SPLINE
SPL {X  -133.093, Y  +296.896, Z    +0.000, E1   +44.059, E3 +170338.505}
SPL {X  -150.601, Y  +331.670, Z    +0.000, E1   +33.435, E3 +170362.768}
SPL {X  -157.739, Y  +358.898, Z    +0.000, E1   +20.026, E3 +170370.995}
SPL {X  -159.601, Y  +374.403, Z    +0.000, E1   +10.058, E3 +170373.311}
SPL {X  -159.993, Y  +384.251, Z    +0.000, E1    +2.830, E3 +170373.943}
SPL {X  -160.000, Y  +387.929, Z    +0.000, E1    -0.363, E3 +170374.011}
SPL {X  -160.000, Y  +392.137, Z    +0.000, E1    -6.580, E3 +170374.150}
SPL {X  -160.000, Y  +398.334, Z    +0.000, E1   -17.404, E3 +170374.642}
SPL {X  -160.000, Y  +410.558, Z    +0.000, E1   -36.649, E3 +170376.745}
SPL {X  -160.000, Y  +459.534, Z    +0.000, E1   -61.429, E3 +170396.339}
SPL {X  -160.000, Y  +586.246, Z    +0.000, E1   -66.315, E3 +170482.839}
SPL {X  -160.000, Y  +602.823, Z    +0.000, E1   -66.332, E3 +170498.243}
SPL {X  -160.000, Y  +621.796, Z    +0.000, E1   -66.332, E3 +170515.912}
SPL {X  -160.000, Y  +638.226, Z    +0.000, E1   -66.314, E3 +170531.239}
SPL {X  -160.000, Y  +655.092, Z    +0.000, E1   -66.336, E3 +170546.898}
SPL {X  -160.000, Y  +671.716, Z    +0.000, E1   -66.315, E3 +170562.412}
SPL {X  -159.502, Y  +687.017, Z    +0.000, E1   -66.266, E3 +170577.162}
SPL {X  -157.713, Y  +701.353, Z    +0.000, E1   -66.026, E3 +170592.389}
SPL {X  -155.081, Y  +713.767, Z    +0.000, E1   -65.665, E3 +170606.674}
SPL {X  -152.128, Y  +723.968, Z    +0.000, E1   -65.242, E3 +170619.174}
SPL {X  -148.925, Y  +732.892, Z    +0.000, E1   -64.779, E3 +170630.674}
SPL {X  -144.887, Y  +742.280, Z    +0.000, E1   -64.184, E3 +170643.303}
SPL {X  -140.317, Y  +751.285, Z    +0.000, E1   -63.454, E3 +170655.941}
SPL {X  -135.706, Y  +759.158, Z    +0.000, E1   -62.682, E3 +170667.342}
SPL {X  -131.040, Y  +766.207, Z    +0.000, E1   -61.854, E3 +170677.774}
SPL {X  -102.962, Y  +796.870, Z    +0.000, E1   -51.620, E3 +170803.106}
ENDSPLINE

SPLINE
SPL {X  -139.855, Y  +752.122, Z    +0.000, E1   -42.075, E3 +170926.034}
SPL {X  -153.268, Y  +720.324, Z    +0.000, E1   -30.648, E3 +170942.280}
SPL {X  -158.910, Y  +693.048, Z    +0.000, E1   -15.531, E3 +170948.350}
SPL {X  -159.977, Y  +677.095, Z    +0.000, E1    -3.968, E3 +170949.774}
SPL {X  -160.000, Y  +672.556, Z    +0.000, E1    -0.073, E3 +170949.876}
SPL {X  -160.000, Y  +669.399, Z    +0.000, E1    +3.976, E3 +170949.956}
SPL {X  -160.000, Y  +661.045, Z    +0.000, E1   +19.300, E3 +170950.544}
SPL {X  -160.000, Y  +646.999, Z    +0.000, E1   +41.048, E3 +170952.962}
SPL {X  -160.000, Y  +594.464, Z    +0.000, E1   +63.651, E3 +170973.262}
SPL {X  -160.000, Y  +465.200, Z    +0.000, E1   +67.027, E3 +171061.832}
SPL {X  -160.000, Y  +444.745, Z    +0.000, E1   +67.032, E3 +171080.241}
SPL {X  -160.000, Y  +422.224, Z    +0.000, E1   +67.044, E3 +171100.493}
ENDSPLINE

SPLINE
SPL {X  -160.000, Y  +424.635, Z    +0.000, E1   +64.425, E3 +171118.519}
ENDSPLINE

SPLINE
SPL {X  -160.000, Y  +410.501, Z    +0.000, E1   +64.162, E3 +171135.064}
SPL {X  -160.000, Y  +387.965, Z    +0.000, E1   +65.039, E3 +171151.016}
SPL {X  -158.836, Y  +366.435, Z    +0.000, E1   +65.805, E3 +171165.957}
SPL {X  -155.922, Y  +349.806, Z    +0.000, E1   +65.927, E3 +171180.603}
SPL {X  -152.875, Y  +338.486, Z    +0.000, E1   +65.488, E3 +171194.220}
SPL {X  -149.360, Y  +328.327, Z    +0.000, E1   +64.994, E3 +171207.126}
SPL {X  -145.195, Y  +318.481, Z    +0.000, E1   +64.365, E3 +171220.280}
SPL {X  -140.564, Y  +309.268, Z    +0.000, E1   +63.646, E3 +171233.101}
SPL {X  -135.770, Y  +301.044, Z    +0.000, E1   +62.840, E3 +171244.972}
SPL {X  -130.944, Y  +293.756, Z    +0.000, E1   +61.990, E3 +171255.715}
SPL {X  -103.957, Y  +264.074, Z    +0.000, E1   +52.557, E3 +171361.819}
ENDSPLINE

SPLINE
SPL {X  -133.093, Y  +296.896, Z    +0.000, E1   +44.059, E3 +171486.653}
SPL {X  -150.601, Y  +331.670, Z    +0.000, E1   +33.435, E3 +171510.915}
SPL {X  -157.739, Y  +358.898, Z    +0.000, E1   +20.026, E3 +171519.143}
SPL {X  -159.601, Y  +374.403, Z    +0.000, E1   +10.058, E3 +171521.459}
SPL {X  -159.993, Y  +384.251, Z    +0.000, E1    +2.830, E3 +171522.091}
SPL {X  -160.000, Y  +387.929, Z    +0.000, E1    -0.363, E3 +171522.159}
SPL {X  -160.000, Y  +392.137, Z    +0.000, E1    -6.580, E3 +171522.298}
SPL {X  -160.000, Y  +398.334, Z    +0.000, E1   -17.404, E3 +171522.790}
SPL {X  -160.000, Y  +410.558, Z    +0.000, E1   -36.649, E3 +171524.893}
SPL {X  -160.000, Y  +459.534, Z    +0.000, E1   -61.429, E3 +171544.487}
SPL {X  -160.000, Y  +586.246, Z    +0.000, E1   -66.315, E3 +171630.987}
SPL {X  -160.000, Y  +602.823, Z    +0.000, E1   -66.332, E3 +171646.391}
SPL {X  -160.000, Y  +621.796, Z    +0.000, E1   -66.332, E3 +171664.060}
SPL {X  -160.000, Y  +638.226, Z    +0.000, E1   -66.314, E3 +171679.387}
SPL {X  -160.000, Y  +655.092, Z    +0.000, E1   -66.336, E3 +171695.046}
SPL {X  -160.000, Y  +671.716, Z    +0.000, E1   -66.315, E3 +171710.560}
SPL {X  -159.502, Y  +687.017, Z    +0.000, E1   -66.266, E3 +171725.310}
SPL {X  -157.713, Y  +701.353, Z    +0.000, E1   -66.026, E3 +171740.537}
SPL {X  -155.081, Y  +713.767, Z    +0.000, E1   -65.665, E3 +171754.822}
SPL {X  -152.128, Y  +723.968, Z    +0.000, E1   -65.242, E3 +171767.322}
SPL {X  -148.925, Y  +732.892, Z    +0.000, E1   -64.779, E3 +171778.822}
SPL {X  -144.887, Y  +742.280, Z    +0.000, E1   -64.184, E3 +171791.451}
SPL {X  -140.317, Y  +751.285, Z    +0.000, E1   -63.454, E3 +171804.089}
SPL {X  -135.706, Y  +759.158, Z    +0.000, E1   -62.682, E3 +171815.490}
SPL {X  -131.040, Y  +766.207, Z    +0.000, E1   -61.854, E3 +171825.922}
SPL {X  -102.962, Y  +796.870, Z    +0.000, E1   -51.620, E3 +171951.254}
ENDSPLINE

SPLINE
SPL {X  -139.855, Y  +752.122, Z    +0.000, E1   -42.075, E3 +172074.182}
SPL {X  -153.268, Y  +720.324, Z    +0.000, E1   -30.648, E3 +172090.427}
SPL {X  -158.910, Y  +693.048, Z    +0.000, E1   -15.531, E3 +172096.498}
SPL {X  -159.977, Y  +677.095, Z    +0.000, E1    -3.968, E3 +172097.922}
SPL {X  -160.000, Y  +672.556, Z    +0.000, E1    -0.073, E3 +172098.024}
SPL {X  -160.000, Y  +669.399, Z    +0.000, E1    +3.976, E3 +172098.104}
SPL {X  -160.000, Y  +661.045, Z    +0.000, E1   +19.300, E3 +172098.692}
SPL {X  -160.000, Y  +646.999, Z    +0.000, E1   +41.048, E3 +172101.110}
SPL {X  -160.000, Y  +594.464, Z    +0.000, E1   +63.651, E3 +172121.410}
SPL {X  -160.000, Y  +465.200, Z    +0.000, E1   +67.027, E3 +172209.980}
SPL {X  -160.000, Y  +444.745, Z    +0.000, E1   +67.032, E3 +172228.389}
SPL {X  -160.000, Y  +422.224, Z    +0.000, E1   +67.044, E3 +172248.641}
ENDSPLINE

SPLINE
SPL {X  -160.000, Y  +424.635, Z    +0.000, E1   +64.425, E3 +172266.667}
ENDSPLINE

SPLINE
SPL {X  -160.000, Y  +410.501, Z    +0.000, E1   +64.162, E3 +172283.212}
SPL {X  -160.000, Y  +387.965, Z    +0.000, E1   +65.039, E3 +172299.163}
SPL {X  -158.836, Y  +366.435, Z    +0.000, E1   +65.805, E3 +172314.105}
SPL {X  -155.922, Y  +349.806, Z    +0.000, E1   +65.927, E3 +172328.751}
SPL {X  -152.875, Y  +338.486, Z    +0.000, E1   +65.488, E3 +172342.368}
SPL {X  -149.360, Y  +328.327, Z    +0.000, E1   +64.994, E3 +172355.274}
SPL {X  -145.195, Y  +318.481, Z    +0.000, E1   +64.365, E3 +172368.428}
SPL {X  -140.564, Y  +309.268, Z    +0.000, E1   +63.646, E3 +172381.249}
SPL {X  -135.770, Y  +301.044, Z    +0.000, E1   +62.840, E3 +172393.120}
SPL {X  -130.944, Y  +293.756, Z    +0.000, E1   +61.990, E3 +172403.863}
SPL {X  -103.957, Y  +264.074, Z    +0.000, E1   +52.557, E3 +172509.967}
ENDSPLINE

SPLINE
SPL {X  -133.093, Y  +296.896, Z    +0.000, E1   +44.059, E3 +172634.801}
SPL {X  -150.601, Y  +331.670, Z    +0.000, E1   +33.435, E3 +172659.063}
SPL {X  -157.739, Y  +358.898, Z    +0.000, E1   +20.026, E3 +172667.291}
SPL {X  -159.601, Y  +374.403, Z    +0.000, E1   +10.058, E3 +172669.607}
SPL {X  -159.993, Y  +384.251, Z    +0.000, E1    +2.830, E3 +172670.239}
SPL {X  -160.000, Y  +387.929, Z    +0.000, E1    -0.363, E3 +172670.307}
SPL {X  -160.000, Y  +392.137, Z    +0.000, E1    -6.580, E3 +172670.446}
SPL {X  -160.000, Y  +398.334, Z    +0.000, E1   -17.404, E3 +172670.938}
SPL {X  -160.000, Y  +410.558, Z    +0.000, E1   -36.649, E3 +172673.041}
SPL {X  -160.000, Y  +459.534, Z    +0.000, E1   -61.429, E3 +172692.635}
SPL {X  -160.000, Y  +586.246, Z    +0.000, E1   -66.315, E3 +172779.135}
SPL {X  -160.000, Y  +602.823, Z    +0.000, E1   -66.332, E3 +172794.539}
SPL {X  -160.000, Y  +621.796, Z    +0.000, E1   -66.332, E3 +172812.207}
SPL {X  -160.000, Y  +638.226, Z    +0.000, E1   -66.314, E3 +172827.535}
SPL {X  -160.000, Y  +655.092, Z    +0.000, E1   -66.336, E3 +172843.194}
SPL {X  -160.000, Y  +671.716, Z    +0.000, E1   -66.315, E3 +172858.708}
SPL {X  -159.502, Y  +687.017, Z    +0.000, E1   -66.266, E3 +172873.458}
SPL {X  -157.713, Y  +701.353, Z    +0.000, E1   -66.026, E3 +172888.685}
SPL {X  -155.081, Y  +713.767, Z    +0.000, E1   -65.665, E3 +172902.970}
SPL {X  -152.128, Y  +723.968, Z    +0.000, E1   -65.242, E3 +172915.470}
SPL {X  -148.925, Y  +732.892, Z    +0.000, E1   -64.779, E3 +172926.970}
SPL {X  -144.887, Y  +742.280, Z    +0.000, E1   -64.184, E3 +172939.599}
SPL {X  -140.317, Y  +751.285, Z    +0.000, E1   -63.454, E3 +172952.237}
SPL {X  -135.706, Y  +759.158, Z    +0.000, E1   -62.682, E3 +172963.638}
SPL {X  -131.040, Y  +766.207, Z    +0.000, E1   -61.854, E3 +172974.070}
SPL {X  -102.962, Y  +796.870, Z    +0.000, E1   -51.620, E3 +173099.401}
ENDSPLINE

SPLINE
SPL {X  -139.855, Y  +752.122, Z    +0.000, E1   -42.075, E3 +173222.330}
SPL {X  -153.268, Y  +720.324, Z    +0.000, E1   -30.648, E3 +173238.575}
SPL {X  -158.910, Y  +693.048, Z    +0.000, E1   -15.531, E3 +173244.646}
SPL {X  -159.977, Y  +677.095, Z    +0.000, E1    -3.968, E3 +173246.070}
SPL {X  -160.000, Y  +672.556, Z    +0.000, E1    -0.073, E3 +173246.172}
SPL {X  -160.000, Y  +669.399, Z    +0.000, E1    +3.976, E3 +173246.251}
SPL {X  -160.000, Y  +661.045, Z    +0.000, E1   +19.300, E3 +173246.840}
SPL {X  -160.000, Y  +646.999, Z    +0.000, E1   +41.048, E3 +173249.258}
SPL {X  -160.000, Y  +594.464, Z    +0.000, E1   +63.651, E3 +173269.558}
SPL {X  -160.000, Y  +465.200, Z    +0.000, E1   +67.027, E3 +173358.128}
SPL {X  -160.000, Y  +444.745, Z    +0.000, E1   +67.032, E3 +173376.537}
SPL {X  -160.000, Y  +422.224, Z    +0.000, E1   +67.044, E3 +173396.788}
ENDSPLINE

SPLINE
SPL {X  -160.000, Y  +424.635, Z    +0.000, E1   +64.425, E3 +173414.815}
ENDSPLINE

SPLINE
SPL {X  -160.000, Y  +410.501, Z    +0.000, E1   +64.162, E3 +173431.360}
SPL {X  -160.000, Y  +387.965, Z    +0.000, E1   +65.039, E3 +173447.311}
SPL {X  -158.836, Y  +366.435, Z    +0.000, E1   +65.805, E3 +173462.252}
SPL {X  -155.922, Y  +349.806, Z    +0.000, E1   +65.927, E3 +173476.899}
SPL {X  -152.875, Y  +338.486, Z    +0.000, E1   +65.488, E3 +173490.516}
SPL {X  -149.360, Y  +328.327, Z    +0.000, E1   +64.994, E3 +173503.422}
SPL {X  -145.195, Y  +318.481, Z    +0.000, E1   +64.365, E3 +173516.576}
SPL {X  -140.564, Y  +309.268, Z    +0.000, E1   +63.646, E3 +173529.397}
SPL {X  -135.770, Y  +301.044, Z    +0.000, E1   +62.840, E3 +173541.268}
SPL {X  -130.944, Y  +293.756, Z    +0.000, E1   +61.990, E3 +173552.011}
SPL {X  -103.957, Y  +264.074, Z    +0.000, E1   +52.557, E3 +173658.115}
ENDSPLINE

SPLINE
SPL {X  -133.093, Y  +296.896, Z    +0.000, E1   +44.059, E3 +173782.949}
SPL {X  -150.601, Y  +331.670, Z    +0.000, E1   +33.435, E3 +173807.211}
SPL {X  -157.739, Y  +358.898, Z    +0.000, E1   +20.026, E3 +173815.439}
SPL {X  -159.601, Y  +374.403, Z    +0.000, E1   +10.058, E3 +173817.755}
SPL {X  -159.993, Y  +384.251, Z    +0.000, E1    +2.830, E3 +173818.387}
SPL {X  -160.000, Y  +387.929, Z    +0.000, E1    -0.363, E3 +173818.455}
SPL {X  -160.000, Y  +392.137, Z    +0.000, E1    -6.580, E3 +173818.594}
SPL {X  -160.000, Y  +398.334, Z    +0.000, E1   -17.404, E3 +173819.086}
SPL {X  -160.000, Y  +410.558, Z    +0.000, E1   -36.649, E3 +173821.189}
SPL {X  -160.000, Y  +459.534, Z    +0.000, E1   -61.429, E3 +173840.783}
SPL {X  -160.000, Y  +586.246, Z    +0.000, E1   -66.315, E3 +173927.283}
SPL {X  -160.000, Y  +602.823, Z    +0.000, E1   -66.332, E3 +173942.687}
SPL {X  -160.000, Y  +621.796, Z    +0.000, E1   -66.332, E3 +173960.355}
SPL {X  -160.000, Y  +638.226, Z    +0.000, E1   -66.314, E3 +173975.683}
SPL {X  -160.000, Y  +655.092, Z    +0.000, E1   -66.336, E3 +173991.342}
SPL {X  -160.000, Y  +671.716, Z    +0.000, E1   -66.315, E3 +174006.855}
SPL {X  -159.502, Y  +687.017, Z    +0.000, E1   -66.266, E3 +174021.606}
SPL {X  -157.713, Y  +701.353, Z    +0.000, E1   -66.026, E3 +174036.833}
SPL {X  -155.081, Y  +713.767, Z    +0.000, E1   -65.665, E3 +174051.118}
SPL {X  -152.128, Y  +723.968, Z    +0.000, E1   -65.242, E3 +174063.618}
SPL {X  -148.925, Y  +732.892, Z    +0.000, E1   -64.779, E3 +174075.118}
SPL {X  -144.887, Y  +742.280, Z    +0.000, E1   -64.184, E3 +174087.747}
SPL {X  -140.317, Y  +751.285, Z    +0.000, E1   -63.454, E3 +174100.385}
SPL {X  -135.706, Y  +759.158, Z    +0.000, E1   -62.682, E3 +174111.786}
SPL {X  -131.040, Y  +766.207, Z    +0.000, E1   -61.854, E3 +174122.217}
SPL {X  -102.962, Y  +796.870, Z    +0.000, E1   -51.620, E3 +174247.549}
ENDSPLINE

SPLINE
SPL {X  -139.855, Y  +752.122, Z    +0.000, E1   -42.075, E3 +174370.478}
SPL {X  -153.268, Y  +720.324, Z    +0.000, E1   -30.648, E3 +174386.723}
SPL {X  -158.910, Y  +693.048, Z    +0.000, E1   -15.531, E3 +174392.794}
SPL {X  -159.977, Y  +677.095, Z    +0.000, E1    -3.968, E3 +174394.218}
SPL {X  -160.000, Y  +672.556, Z    +0.000, E1    -0.073, E3 +174394.320}
SPL {X  -160.000, Y  +669.399, Z    +0.000, E1    +3.976, E3 +174394.399}
SPL {X  -160.000, Y  +661.045, Z    +0.000, E1   +19.300, E3 +174394.988}
SPL {X  -160.000, Y  +646.999, Z    +0.000, E1   +41.048, E3 +174397.406}
SPL {X  -160.000, Y  +594.464, Z    +0.000, E1   +63.651, E3 +174417.706}
SPL {X  -160.000, Y  +465.200, Z    +0.000, E1   +67.027, E3 +174506.276}
SPL {X  -160.000, Y  +444.745, Z    +0.000, E1   +67.032, E3 +174524.685}
SPL {X  -160.000, Y  +422.224, Z    +0.000, E1   +67.044, E3 +174544.936}
ENDSPLINE

SPLINE
SPL {X  -160.000, Y  +424.635, Z    +0.000, E1   +64.425, E3 +174562.963}
ENDSPLINE

SPLINE
SPL {X  -160.000, Y  +410.501, Z    +0.000, E1   +64.162, E3 +174579.508}
SPL {X  -160.000, Y  +387.965, Z    +0.000, E1   +65.039, E3 +174595.459}
SPL {X  -158.836, Y  +366.435, Z    +0.000, E1   +65.805, E3 +174610.400}
ENDSPLINE

SPLINE
SPL {X  -158.528, Y  +364.045, Z    +0.000, E1   +63.714, E3 +174628.761}
SPL {X  -155.923, Y  +349.812, Z    +0.000, E1   +63.321, E3 +174646.317}
SPL {X  -152.732, Y  +338.026, Z    +0.000, E1   +62.842, E3 +174661.851}
SPL {X  -149.257, Y  +328.060, Z    +0.000, E1   +62.292, E3 +174675.708}
SPL {X  -144.838, Y  +317.715, Z    +0.000, E1   +61.617, E3 +174690.714}
SPL {X  -139.661, Y  +307.631, Z    +0.000, E1   +60.727, E3 +174706.017}
SPL {X  -134.254, Y  +298.660, Z    +0.000, E1   +59.757, E3 +174720.065}
SPL {X  -111.782, Y  +271.224, Z    +0.000, E1   +50.030, E3 +174838.488}
ENDSPLINE

SPLINE
SPL {X  -142.230, Y  +312.416, Z    +0.000, E1   +39.081, E3 +174947.609}
SPL {X  -154.023, Y  +342.375, Z    +0.000, E1   +27.770, E3 +174964.066}
SPL {X  -159.227, Y  +369.989, Z    +0.000, E1   +12.792, E3 +174970.758}
SPL {X  -159.997, Y  +384.682, Z    +0.000, E1    +2.433, E3 +174972.123}
SPL {X  -160.000, Y  +388.025, Z    +0.000, E1    -0.434, E3 +174972.193}
SPL {X  -160.000, Y  +391.999, Z    +0.000, E1    -5.822, E3 +174972.338}
SPL {X  -160.000, Y  +397.968, Z    +0.000, E1   -15.492, E3 +174972.852}
SPL {X  -160.000, Y  +409.894, Z    +0.000, E1   -33.660, E3 +174974.960}
SPL {X  -160.000, Y  +457.050, Z    +0.000, E1   -59.500, E3 +174994.156}
SPL {X  -160.000, Y  +570.419, Z    +0.000, E1   -64.293, E3 +175079.721}
SPL {X  -160.000, Y  +587.690, Z    +0.000, E1   -64.299, E3 +175097.384}
SPL {X  -160.000, Y  +605.383, Z    +0.000, E1   -64.296, E3 +175115.482}
SPL {X  -160.000, Y  +621.010, Z    +0.000, E1   -64.279, E3 +175131.492}
SPL {X  -160.000, Y  +636.410, Z    +0.000, E1   -64.294, E3 +175147.221}
SPL {X  -160.000, Y  +654.238, Z    +0.000, E1   -64.301, E3 +175165.426}
SPL {X  -160.000, Y  +670.465, Z    +0.000, E1   -64.283, E3 +175182.050}
SPL {X  -159.617, Y  +685.462, Z    +0.000, E1   -64.244, E3 +175197.777}
SPL {X  -158.001, Y  +699.614, Z    +0.000, E1   -64.013, E3 +175213.952}
SPL {X  -155.628, Y  +711.546, Z    +0.000, E1   -63.666, E3 +175228.621}
SPL {X  -152.846, Y  +721.708, Z    +0.000, E1   -63.251, E3 +175241.854}
SPL {X  -149.418, Y  +731.620, Z    +0.000, E1   -62.736, E3 +175255.409}
SPL {X  -145.585, Y  +740.770, Z    +0.000, E1   -62.119, E3 +175268.507}
SPL {X  -141.572, Y  +748.948, Z    +0.000, E1   -61.453, E3 +175280.632}
SPL {X  -137.548, Y  +756.134, Z    +0.000, E1   -60.743, E3 +175291.641}
SPL {X  -133.391, Y  +762.756, Z    +0.000, E1   -59.994, E3 +175301.958}
SPL {X  -109.419, Y  +791.137, Z    +0.000, E1   -49.920, E3 +175435.247}
ENDSPLINE

SPLINE
SPL {X  -148.079, Y  +735.002, Z    +0.000, E1   -35.426, E3 +175542.830}
SPL {X  -158.158, Y  +698.608, Z    +0.000, E1   -18.222, E3 +175555.483}
SPL {X  -159.870, Y  +680.839, Z    +0.000, E1    -6.577, E3 +175557.870}
SPL {X  -160.000, Y  +671.754, Z    +0.000, E1    +0.400, E3 +175558.229}
SPL {X  -160.000, Y  +663.703, Z    +0.000, E1   +12.763, E3 +175558.695}
SPL {X  -160.000, Y  +653.310, Z    +0.000, E1   +30.441, E3 +175560.165}
SPL {X  -160.000, Y  +640.945, Z    +0.000, E1   +44.811, E3 +175563.377}
SPL {X  -160.000, Y  +592.314, Z    +0.000, E1   +61.740, E3 +175585.371}
SPL {X  -160.000, Y  +478.009, Z    +0.000, E1   +65.091, E3 +175672.428}
SPL {X  -160.000, Y  +417.917, Z    +0.000, E1   +69.146, E3 +175692.599}
SPL {X  -160.000, Y  +403.867, Z    +0.000, E1   +68.803, E3 +175707.091}
SPL {X  -160.000, Y  +399.669, Z    +0.000, E1   +67.598, E3 +175720.962}
SPL {X  -160.000, Y  +392.628, Z    +0.000, E1   +66.554, E3 +175735.993}
SPL {X  -159.998, Y  +384.859, Z    +0.000, E1   +65.356, E3 +175752.921}
SPL {X  -159.712, Y  +376.098, Z    +0.000, E1   +64.333, E3 +175769.466}
SPL {X  -158.506, Y  +363.887, Z    +0.000, E1   +63.706, E3 +175786.858}
SPL {X  -155.923, Y  +349.812, Z    +0.000, E1   +63.321, E3 +175804.211}
SPL {X  -152.732, Y  +338.026, Z    +0.000, E1   +62.842, E3 +175819.746}
SPL {X  -149.257, Y  +328.060, Z    +0.000, E1   +62.292, E3 +175833.602}
SPL {X  -144.838, Y  +317.715, Z    +0.000, E1   +61.617, E3 +175848.608}
SPL {X  -139.661, Y  +307.631, Z    +0.000, E1   +60.727, E3 +175863.911}
SPL {X  -134.254, Y  +298.660, Z    +0.000, E1   +59.757, E3 +175877.960}
SPL {X  -111.782, Y  +271.224, Z    +0.000, E1   +50.030, E3 +175996.383}
ENDSPLINE

SPLINE
SPL {X  -142.230, Y  +312.416, Z    +0.000, E1   +39.081, E3 +176105.503}
SPL {X  -154.023, Y  +342.375, Z    +0.000, E1   +27.770, E3 +176121.960}
SPL {X  -159.227, Y  +369.989, Z    +0.000, E1   +12.792, E3 +176128.653}
SPL {X  -159.997, Y  +384.682, Z    +0.000, E1    +2.433, E3 +176130.018}
SPL {X  -160.000, Y  +388.025, Z    +0.000, E1    -0.434, E3 +176130.088}
SPL {X  -160.000, Y  +391.999, Z    +0.000, E1    -5.822, E3 +176130.233}
SPL {X  -160.000, Y  +397.968, Z    +0.000, E1   -15.492, E3 +176130.747}
SPL {X  -160.000, Y  +409.894, Z    +0.000, E1   -33.660, E3 +176132.854}
SPL {X  -160.000, Y  +457.050, Z    +0.000, E1   -59.500, E3 +176152.051}
SPL {X  -160.000, Y  +570.419, Z    +0.000, E1   -64.293, E3 +176237.615}
SPL {X  -160.000, Y  +587.690, Z    +0.000, E1   -64.299, E3 +176255.278}
SPL {X  -160.000, Y  +605.383, Z    +0.000, E1   -64.296, E3 +176273.376}
SPL {X  -160.000, Y  +621.010, Z    +0.000, E1   -64.279, E3 +176289.386}
SPL {X  -160.000, Y  +636.410, Z    +0.000, E1   -64.294, E3 +176305.115}
SPL {X  -160.000, Y  +654.238, Z    +0.000, E1   -64.301, E3 +176323.321}
SPL {X  -160.000, Y  +670.465, Z    +0.000, E1   -64.283, E3 +176339.944}
SPL {X  -159.617, Y  +685.462, Z    +0.000, E1   -64.244, E3 +176355.672}
SPL {X  -158.001, Y  +699.614, Z    +0.000, E1   -64.013, E3 +176371.847}
SPL {X  -155.628, Y  +711.546, Z    +0.000, E1   -63.666, E3 +176386.516}
SPL {X  -152.846, Y  +721.708, Z    +0.000, E1   -63.251, E3 +176399.749}
SPL {X  -149.418, Y  +731.620, Z    +0.000, E1   -62.736, E3 +176413.303}
SPL {X  -145.585, Y  +740.770, Z    +0.000, E1   -62.119, E3 +176426.402}
SPL {X  -141.572, Y  +748.948, Z    +0.000, E1   -61.453, E3 +176438.526}
SPL {X  -137.548, Y  +756.134, Z    +0.000, E1   -60.743, E3 +176449.536}
SPL {X  -133.391, Y  +762.756, Z    +0.000, E1   -59.994, E3 +176459.852}
SPL {X  -109.419, Y  +791.137, Z    +0.000, E1   -49.920, E3 +176593.141}
ENDSPLINE

SPLINE
SPL {X  -148.079, Y  +735.002, Z    +0.000, E1   -35.426, E3 +176700.724}
SPL {X  -158.158, Y  +698.608, Z    +0.000, E1   -18.222, E3 +176713.377}
SPL {X  -159.870, Y  +680.839, Z    +0.000, E1    -6.577, E3 +176715.765}
SPL {X  -160.000, Y  +671.754, Z    +0.000, E1    +0.400, E3 +176716.123}
SPL {X  -160.000, Y  +663.703, Z    +0.000, E1   +12.763, E3 +176716.589}
SPL {X  -160.000, Y  +653.310, Z    +0.000, E1   +30.441, E3 +176718.059}
SPL {X  -160.000, Y  +640.945, Z    +0.000, E1   +44.811, E3 +176721.271}
SPL {X  -160.000, Y  +592.314, Z    +0.000, E1   +61.740, E3 +176743.265}
SPL {X  -160.000, Y  +478.009, Z    +0.000, E1   +65.091, E3 +176830.323}
SPL {X  -160.000, Y  +417.917, Z    +0.000, E1   +69.146, E3 +176850.493}
SPL {X  -160.000, Y  +403.867, Z    +0.000, E1   +68.803, E3 +176864.985}
SPL {X  -160.000, Y  +399.669, Z    +0.000, E1   +67.598, E3 +176878.857}
SPL {X  -160.000, Y  +392.628, Z    +0.000, E1   +66.554, E3 +176893.887}
SPL {X  -159.998, Y  +384.859, Z    +0.000, E1   +65.356, E3 +176910.816}
SPL {X  -159.712, Y  +376.098, Z    +0.000, E1   +64.333, E3 +176927.360}
SPL {X  -158.506, Y  +363.887, Z    +0.000, E1   +63.706, E3 +176944.752}
SPL {X  -155.923, Y  +349.812, Z    +0.000, E1   +63.321, E3 +176962.105}
SPL {X  -152.732, Y  +338.026, Z    +0.000, E1   +62.842, E3 +176977.640}
SPL {X  -149.257, Y  +328.060, Z    +0.000, E1   +62.292, E3 +176991.497}
SPL {X  -144.838, Y  +317.715, Z    +0.000, E1   +61.617, E3 +177006.502}
SPL {X  -139.661, Y  +307.631, Z    +0.000, E1   +60.727, E3 +177021.806}
SPL {X  -134.254, Y  +298.660, Z    +0.000, E1   +59.757, E3 +177035.854}
SPL {X  -111.782, Y  +271.224, Z    +0.000, E1   +50.030, E3 +177154.277}
ENDSPLINE

SPLINE
SPL {X  -142.230, Y  +312.416, Z    +0.000, E1   +39.081, E3 +177263.397}
SPL {X  -154.023, Y  +342.375, Z    +0.000, E1   +27.770, E3 +177279.854}
SPL {X  -159.227, Y  +369.989, Z    +0.000, E1   +12.792, E3 +177286.547}
SPL {X  -159.997, Y  +384.682, Z    +0.000, E1    +2.433, E3 +177287.912}
SPL {X  -160.000, Y  +388.025, Z    +0.000, E1    -0.434, E3 +177287.982}
SPL {X  -160.000, Y  +391.999, Z    +0.000, E1    -5.822, E3 +177288.127}
SPL {X  -160.000, Y  +397.968, Z    +0.000, E1   -15.492, E3 +177288.641}
SPL {X  -160.000, Y  +409.894, Z    +0.000, E1   -33.660, E3 +177290.748}
SPL {X  -160.000, Y  +457.050, Z    +0.000, E1   -59.500, E3 +177309.945}
SPL {X  -160.000, Y  +570.419, Z    +0.000, E1   -64.293, E3 +177395.510}
SPL {X  -160.000, Y  +587.690, Z    +0.000, E1   -64.299, E3 +177413.172}
SPL {X  -160.000, Y  +605.383, Z    +0.000, E1   -64.296, E3 +177431.271}
SPL {X  -160.000, Y  +621.010, Z    +0.000, E1   -64.279, E3 +177447.281}
SPL {X  -160.000, Y  +636.410, Z    +0.000, E1   -64.294, E3 +177463.009}
SPL {X  -160.000, Y  +654.238, Z    +0.000, E1   -64.301, E3 +177481.215}
SPL {X  -160.000, Y  +670.465, Z    +0.000, E1   -64.283, E3 +177497.838}
SPL {X  -159.617, Y  +685.462, Z    +0.000, E1   -64.244, E3 +177513.566}
SPL {X  -158.001, Y  +699.614, Z    +0.000, E1   -64.013, E3 +177529.741}
SPL {X  -155.628, Y  +711.546, Z    +0.000, E1   -63.666, E3 +177544.410}
SPL {X  -152.846, Y  +721.708, Z    +0.000, E1   -63.251, E3 +177557.643}
SPL {X  -149.418, Y  +731.620, Z    +0.000, E1   -62.736, E3 +177571.197}
SPL {X  -145.585, Y  +740.770, Z    +0.000, E1   -62.119, E3 +177584.296}
SPL {X  -141.572, Y  +748.948, Z    +0.000, E1   -61.453, E3 +177596.420}
SPL {X  -137.548, Y  +756.134, Z    +0.000, E1   -60.743, E3 +177607.430}
SPL {X  -133.391, Y  +762.756, Z    +0.000, E1   -59.994, E3 +177617.747}
SPL {X  -109.419, Y  +791.137, Z    +0.000, E1   -49.920, E3 +177751.036}
ENDSPLINE

SPLINE
SPL {X  -148.079, Y  +735.002, Z    +0.000, E1   -35.426, E3 +177858.618}
SPL {X  -158.158, Y  +698.608, Z    +0.000, E1   -18.222, E3 +177871.271}
SPL {X  -159.870, Y  +680.839, Z    +0.000, E1    -6.577, E3 +177873.659}
SPL {X  -160.000, Y  +671.754, Z    +0.000, E1    +0.400, E3 +177874.018}
SPL {X  -160.000, Y  +663.703, Z    +0.000, E1   +12.763, E3 +177874.483}
SPL {X  -160.000, Y  +653.310, Z    +0.000, E1   +30.441, E3 +177875.954}
SPL {X  -160.000, Y  +640.945, Z    +0.000, E1   +44.811, E3 +177879.166}
SPL {X  -160.000, Y  +592.314, Z    +0.000, E1   +61.740, E3 +177901.159}
SPL {X  -160.000, Y  +478.009, Z    +0.000, E1   +65.091, E3 +177988.217}
SPL {X  -160.000, Y  +417.917, Z    +0.000, E1   +69.146, E3 +178008.387}
SPL {X  -160.000, Y  +403.867, Z    +0.000, E1   +68.803, E3 +178022.880}
SPL {X  -160.000, Y  +399.669, Z    +0.000, E1   +67.598, E3 +178036.751}
SPL {X  -160.000, Y  +392.628, Z    +0.000, E1   +66.554, E3 +178051.782}
SPL {X  -159.998, Y  +384.859, Z    +0.000, E1   +65.356, E3 +178068.710}
SPL {X  -159.712, Y  +376.098, Z    +0.000, E1   +64.333, E3 +178085.255}
SPL {X  -158.506, Y  +363.887, Z    +0.000, E1   +63.706, E3 +178102.647}
SPL {X  -155.923, Y  +349.812, Z    +0.000, E1   +63.321, E3 +178120.000}
SPL {X  -152.732, Y  +338.026, Z    +0.000, E1   +62.842, E3 +178135.534}
SPL {X  -149.257, Y  +328.060, Z    +0.000, E1   +62.292, E3 +178149.391}
SPL {X  -144.838, Y  +317.715, Z    +0.000, E1   +61.617, E3 +178164.397}
SPL {X  -139.661, Y  +307.631, Z    +0.000, E1   +60.727, E3 +178179.700}
SPL {X  -134.254, Y  +298.660, Z    +0.000, E1   +59.757, E3 +178193.748}
SPL {X  -111.782, Y  +271.224, Z    +0.000, E1   +50.030, E3 +178312.171}
ENDSPLINE

SPLINE
SPL {X  -142.230, Y  +312.416, Z    +0.000, E1   +39.081, E3 +178421.292}
SPL {X  -154.023, Y  +342.375, Z    +0.000, E1   +27.770, E3 +178437.749}
SPL {X  -159.227, Y  +369.989, Z    +0.000, E1   +12.792, E3 +178444.441}
SPL {X  -159.997, Y  +384.682, Z    +0.000, E1    +2.433, E3 +178445.806}
SPL {X  -160.000, Y  +388.025, Z    +0.000, E1    -0.434, E3 +178445.876}
SPL {X  -160.000, Y  +391.999, Z    +0.000, E1    -5.822, E3 +178446.021}
SPL {X  -160.000, Y  +397.968, Z    +0.000, E1   -15.492, E3 +178446.535}
SPL {X  -160.000, Y  +409.894, Z    +0.000, E1   -33.660, E3 +178448.643}
SPL {X  -160.000, Y  +457.050, Z    +0.000, E1   -59.500, E3 +178467.839}
SPL {X  -160.000, Y  +570.419, Z    +0.000, E1   -64.293, E3 +178553.404}
SPL {X  -160.000, Y  +587.690, Z    +0.000, E1   -64.299, E3 +178571.067}
SPL {X  -160.000, Y  +605.383, Z    +0.000, E1   -64.296, E3 +178589.165}
SPL {X  -160.000, Y  +621.010, Z    +0.000, E1   -64.279, E3 +178605.175}
SPL {X  -160.000, Y  +636.410, Z    +0.000, E1   -64.294, E3 +178620.904}
SPL {X  -160.000, Y  +654.238, Z    +0.000, E1   -64.301, E3 +178639.109}
SPL {X  -160.000, Y  +670.465, Z    +0.000, E1   -64.283, E3 +178655.733}
SPL {X  -159.617, Y  +685.462, Z    +0.000, E1   -64.244, E3 +178671.460}
SPL {X  -158.001, Y  +699.614, Z    +0.000, E1   -64.013, E3 +178687.635}
SPL {X  -155.628, Y  +711.546, Z    +0.000, E1   -63.666, E3 +178702.304}
SPL {X  -152.846, Y  +721.708, Z    +0.000, E1   -63.251, E3 +178715.537}
SPL {X  -149.418, Y  +731.620, Z    +0.000, E1   -62.736, E3 +178729.092}
SPL {X  -145.585, Y  +740.770, Z    +0.000, E1   -62.119, E3 +178742.190}
SPL {X  -141.572, Y  +748.948, Z    +0.000, E1   -61.453, E3 +178754.315}
SPL {X  -137.548, Y  +756.134, Z    +0.000, E1   -60.743, E3 +178765.324}
SPL {X  -133.391, Y  +762.756, Z    +0.000, E1   -59.994, E3 +178775.641}
SPL {X  -109.419, Y  +791.137, Z    +0.000, E1   -49.920, E3 +178908.930}
ENDSPLINE

SPLINE
SPL {X  -148.079, Y  +735.002, Z    +0.000, E1   -35.426, E3 +179016.512}
SPL {X  -158.158, Y  +698.608, Z    +0.000, E1   -18.222, E3 +179029.166}
SPL {X  -159.870, Y  +680.839, Z    +0.000, E1    -6.577, E3 +179031.553}
SPL {X  -160.000, Y  +671.754, Z    +0.000, E1    +0.400, E3 +179031.912}
SPL {X  -160.000, Y  +663.703, Z    +0.000, E1   +12.763, E3 +179032.378}
SPL {X  -160.000, Y  +653.310, Z    +0.000, E1   +30.441, E3 +179033.848}
SPL {X  -160.000, Y  +640.945, Z    +0.000, E1   +44.811, E3 +179037.060}
SPL {X  -160.000, Y  +592.314, Z    +0.000, E1   +61.740, E3 +179059.054}
SPL {X  -160.000, Y  +478.009, Z    +0.000, E1   +65.091, E3 +179146.111}
SPL {X  -160.000, Y  +417.917, Z    +0.000, E1   +69.146, E3 +179166.281}
SPL {X  -160.000, Y  +403.867, Z    +0.000, E1   +68.803, E3 +179180.774}
SPL {X  -160.000, Y  +399.669, Z    +0.000, E1   +67.598, E3 +179194.645}
SPL {X  -160.000, Y  +392.628, Z    +0.000, E1   +66.554, E3 +179209.676}
SPL {X  -159.998, Y  +384.859, Z    +0.000, E1   +65.356, E3 +179226.604}
SPL {X  -159.712, Y  +376.098, Z    +0.000, E1   +64.333, E3 +179243.149}
SPL {X  -158.506, Y  +363.887, Z    +0.000, E1   +63.706, E3 +179260.541}
SPL {X  -155.923, Y  +349.812, Z    +0.000, E1   +63.321, E3 +179277.894}
SPL {X  -152.732, Y  +338.026, Z    +0.000, E1   +62.842, E3 +179293.429}
SPL {X  -149.257, Y  +328.060, Z    +0.000, E1   +62.292, E3 +179307.285}
SPL {X  -144.838, Y  +317.715, Z    +0.000, E1   +61.617, E3 +179322.291}
SPL {X  -139.661, Y  +307.631, Z    +0.000, E1   +60.727, E3 +179337.594}
SPL {X  -134.254, Y  +298.660, Z    +0.000, E1   +59.757, E3 +179351.643}
SPL {X  -111.782, Y  +271.224, Z    +0.000, E1   +50.030, E3 +179470.066}
ENDSPLINE

SPLINE
SPL {X  -142.230, Y  +312.416, Z    +0.000, E1   +39.081, E3 +179579.186}
SPL {X  -154.023, Y  +342.375, Z    +0.000, E1   +27.770, E3 +179595.643}
SPL {X  -159.227, Y  +369.989, Z    +0.000, E1   +12.792, E3 +179602.336}
SPL {X  -159.997, Y  +384.682, Z    +0.000, E1    +2.433, E3 +179603.701}
SPL {X  -160.000, Y  +388.025, Z    +0.000, E1    -0.434, E3 +179603.771}
SPL {X  -160.000, Y  +391.999, Z    +0.000, E1    -5.822, E3 +179603.916}
SPL {X  -160.000, Y  +397.968, Z    +0.000, E1   -15.492, E3 +179604.430}
SPL {X  -160.000, Y  +409.894, Z    +0.000, E1   -33.660, E3 +179606.537}
SPL {X  -160.000, Y  +457.050, Z    +0.000, E1   -59.500, E3 +179625.733}
SPL {X  -160.000, Y  +570.419, Z    +0.000, E1   -64.293, E3 +179711.298}
SPL {X  -160.000, Y  +587.690, Z    +0.000, E1   -64.299, E3 +179728.961}
SPL {X  -160.000, Y  +605.383, Z    +0.000, E1   -64.296, E3 +179747.059}
SPL {X  -160.000, Y  +621.010, Z    +0.000, E1   -64.279, E3 +179763.069}
SPL {X  -160.000, Y  +636.410, Z    +0.000, E1   -64.294, E3 +179778.798}
SPL {X  -160.000, Y  +654.238, Z    +0.000, E1   -64.301, E3 +179797.004}
SPL {X  -160.000, Y  +670.465, Z    +0.000, E1   -64.283, E3 +179813.627}
SPL {X  -159.617, Y  +685.462, Z    +0.000, E1   -64.244, E3 +179829.355}
SPL {X  -158.001, Y  +699.614, Z    +0.000, E1   -64.013, E3 +179845.530}
SPL {X  -155.628, Y  +711.546, Z    +0.000, E1   -63.666, E3 +179860.199}
SPL {X  -152.846, Y  +721.708, Z    +0.000, E1   -63.251, E3 +179873.432}
SPL {X  -149.418, Y  +731.620, Z    +0.000, E1   -62.736, E3 +179886.986}
SPL {X  -145.585, Y  +740.770, Z    +0.000, E1   -62.119, E3 +179900.085}
SPL {X  -141.572, Y  +748.948, Z    +0.000, E1   -61.453, E3 +179912.209}
SPL {X  -137.548, Y  +756.134, Z    +0.000, E1   -60.743, E3 +179923.219}
SPL {X  -133.391, Y  +762.756, Z    +0.000, E1   -59.994, E3 +179933.535}
SPL {X  -109.419, Y  +791.137, Z    +0.000, E1   -49.920, E3 +180066.824}
ENDSPLINE

SPLINE
SPL {X  -148.079, Y  +735.002, Z    +0.000, E1   -35.426, E3 +180174.407}
SPL {X  -158.158, Y  +698.608, Z    +0.000, E1   -18.222, E3 +180187.060}
SPL {X  -159.870, Y  +680.839, Z    +0.000, E1    -6.577, E3 +180189.448}
SPL {X  -160.000, Y  +671.754, Z    +0.000, E1    +0.400, E3 +180189.806}
SPL {X  -160.000, Y  +663.703, Z    +0.000, E1   +12.763, E3 +180190.272}
SPL {X  -160.000, Y  +653.310, Z    +0.000, E1   +30.441, E3 +180191.742}
SPL {X  -160.000, Y  +640.945, Z    +0.000, E1   +44.811, E3 +180194.954}
SPL {X  -160.000, Y  +592.314, Z    +0.000, E1   +61.740, E3 +180216.948}
SPL {X  -160.000, Y  +478.009, Z    +0.000, E1   +65.091, E3 +180304.006}
SPL {X  -160.000, Y  +417.917, Z    +0.000, E1   +69.146, E3 +180324.176}
SPL {X  -160.000, Y  +403.867, Z    +0.000, E1   +68.803, E3 +180338.668}
SPL {X  -160.000, Y  +399.669, Z    +0.000, E1   +67.598, E3 +180352.540}
SPL {X  -160.000, Y  +392.628, Z    +0.000, E1   +66.554, E3 +180367.570}
SPL {X  -159.998, Y  +384.859, Z    +0.000, E1   +65.356, E3 +180384.499}
SPL {X  -159.712, Y  +376.098, Z    +0.000, E1   +64.333, E3 +180401.043}
SPL {X  -158.506, Y  +363.887, Z    +0.000, E1   +63.706, E3 +180418.435}
SPL {X  -155.923, Y  +349.812, Z    +0.000, E1   +63.321, E3 +180435.788}
SPL {X  -152.732, Y  +338.026, Z    +0.000, E1   +62.842, E3 +180451.323}
SPL {X  -149.257, Y  +328.060, Z    +0.000, E1   +62.292, E3 +180465.180}
SPL {X  -144.838, Y  +317.715, Z    +0.000, E1   +61.617, E3 +180480.185}
SPL {X  -139.661, Y  +307.631, Z    +0.000, E1   +60.727, E3 +180495.489}
SPL {X  -134.254, Y  +298.660, Z    +0.000, E1   +59.757, E3 +180509.537}
SPL {X  -111.782, Y  +271.224, Z    +0.000, E1   +50.030, E3 +180627.960}
ENDSPLINE

SPLINE
SPL {X  -142.230, Y  +312.416, Z    +0.000, E1   +39.081, E3 +180737.080}
SPL {X  -154.023, Y  +342.375, Z    +0.000, E1   +27.770, E3 +180753.537}
SPL {X  -159.227, Y  +369.989, Z    +0.000, E1   +12.792, E3 +180760.230}
SPL {X  -159.997, Y  +384.682, Z    +0.000, E1    +2.433, E3 +180761.595}
SPL {X  -160.000, Y  +388.025, Z    +0.000, E1    -0.434, E3 +180761.665}
SPL {X  -160.000, Y  +391.999, Z    +0.000, E1    -5.822, E3 +180761.810}
SPL {X  -160.000, Y  +397.968, Z    +0.000, E1   -15.492, E3 +180762.324}
SPL {X  -160.000, Y  +409.894, Z    +0.000, E1   -33.660, E3 +180764.431}
SPL {X  -160.000, Y  +457.050, Z    +0.000, E1   -59.500, E3 +180783.628}
SPL {X  -160.000, Y  +570.419, Z    +0.000, E1   -64.293, E3 +180869.193}
SPL {X  -160.000, Y  +587.690, Z    +0.000, E1   -64.299, E3 +180886.855}
SPL {X  -160.000, Y  +605.383, Z    +0.000, E1   -64.296, E3 +180904.953}
SPL {X  -160.000, Y  +621.010, Z    +0.000, E1   -64.279, E3 +180920.964}
SPL {X  -160.000, Y  +636.410, Z    +0.000, E1   -64.294, E3 +180936.692}
SPL {X  -160.000, Y  +654.238, Z    +0.000, E1   -64.301, E3 +180954.898}
SPL {X  -160.000, Y  +670.465, Z    +0.000, E1   -64.283, E3 +180971.521}
SPL {X  -159.617, Y  +685.462, Z    +0.000, E1   -64.244, E3 +180987.249}
SPL {X  -158.001, Y  +699.614, Z    +0.000, E1   -64.013, E3 +181003.424}
SPL {X  -155.628, Y  +711.546, Z    +0.000, E1   -63.666, E3 +181018.093}
SPL {X  -152.846, Y  +721.708, Z    +0.000, E1   -63.251, E3 +181031.326}
SPL {X  -149.418, Y  +731.620, Z    +0.000, E1   -62.736, E3 +181044.880}
SPL {X  -145.585, Y  +740.770, Z    +0.000, E1   -62.119, E3 +181057.979}
SPL {X  -141.572, Y  +748.948, Z    +0.000, E1   -61.453, E3 +181070.103}
SPL {X  -137.548, Y  +756.134, Z    +0.000, E1   -60.743, E3 +181081.113}
SPL {X  -133.391, Y  +762.756, Z    +0.000, E1   -59.994, E3 +181091.429}
SPL {X  -109.419, Y  +791.137, Z    +0.000, E1   -49.920, E3 +181224.719}
ENDSPLINE

SPLINE
SPL {X  -148.079, Y  +735.002, Z    +0.000, E1   -35.426, E3 +181332.301}
SPL {X  -158.158, Y  +698.608, Z    +0.000, E1   -18.222, E3 +181344.954}
SPL {X  -159.870, Y  +680.839, Z    +0.000, E1    -6.577, E3 +181347.342}
SPL {X  -160.000, Y  +671.754, Z    +0.000, E1    +0.400, E3 +181347.701}
SPL {X  -160.000, Y  +663.703, Z    +0.000, E1   +12.763, E3 +181348.166}
SPL {X  -160.000, Y  +653.310, Z    +0.000, E1   +30.441, E3 +181349.636}
SPL {X  -160.000, Y  +640.945, Z    +0.000, E1   +44.811, E3 +181352.849}
SPL {X  -160.000, Y  +592.314, Z    +0.000, E1   +61.740, E3 +181374.842}
SPL {X  -160.000, Y  +478.009, Z    +0.000, E1   +65.091, E3 +181461.900}
SPL {X  -160.000, Y  +417.917, Z    +0.000, E1   +69.146, E3 +181482.070}
SPL {X  -160.000, Y  +403.867, Z    +0.000, E1   +68.803, E3 +181496.563}
SPL {X  -160.000, Y  +399.669, Z    +0.000, E1   +67.598, E3 +181510.434}
SPL {X  -160.000, Y  +392.628, Z    +0.000, E1   +66.554, E3 +181525.465}
SPL {X  -159.998, Y  +384.859, Z    +0.000, E1   +65.356, E3 +181542.393}
SPL {X  -159.712, Y  +376.098, Z    +0.000, E1   +64.333, E3 +181558.938}
SPL {X  -158.506, Y  +363.887, Z    +0.000, E1   +63.706, E3 +181576.330}
SPL {X  -155.923, Y  +349.812, Z    +0.000, E1   +63.321, E3 +181593.683}
SPL {X  -152.732, Y  +338.026, Z    +0.000, E1   +62.842, E3 +181609.217}
SPL {X  -149.257, Y  +328.060, Z    +0.000, E1   +62.292, E3 +181623.074}
SPL {X  -144.838, Y  +317.715, Z    +0.000, E1   +61.617, E3 +181638.080}
SPL {X  -139.661, Y  +307.631, Z    +0.000, E1   +60.727, E3 +181653.383}
SPL {X  -134.254, Y  +298.660, Z    +0.000, E1   +59.757, E3 +181667.431}
SPL {X  -111.782, Y  +271.224, Z    +0.000, E1   +50.030, E3 +181785.854}
ENDSPLINE

SPLINE
SPL {X  -142.230, Y  +312.416, Z    +0.000, E1   +39.081, E3 +181894.975}
SPL {X  -154.023, Y  +342.375, Z    +0.000, E1   +27.770, E3 +181911.431}
SPL {X  -159.227, Y  +369.989, Z    +0.000, E1   +12.792, E3 +181918.124}
SPL {X  -159.997, Y  +384.682, Z    +0.000, E1    +2.433, E3 +181919.489}
SPL {X  -160.000, Y  +388.025, Z    +0.000, E1    -0.434, E3 +181919.559}
SPL {X  -160.000, Y  +391.999, Z    +0.000, E1    -5.822, E3 +181919.704}
SPL {X  -160.000, Y  +397.968, Z    +0.000, E1   -15.492, E3 +181920.218}
SPL {X  -160.000, Y  +409.894, Z    +0.000, E1   -33.660, E3 +181922.326}
SPL {X  -160.000, Y  +457.050, Z    +0.000, E1   -59.500, E3 +181941.522}
SPL {X  -160.000, Y  +570.419, Z    +0.000, E1   -64.293, E3 +182027.087}
SPL {X  -160.000, Y  +587.690, Z    +0.000, E1   -64.299, E3 +182044.749}
SPL {X  -160.000, Y  +605.383, Z    +0.000, E1   -64.296, E3 +182062.848}
SPL {X  -160.000, Y  +621.010, Z    +0.000, E1   -64.279, E3 +182078.858}
SPL {X  -160.000, Y  +636.410, Z    +0.000, E1   -64.294, E3 +182094.587}
SPL {X  -160.000, Y  +654.238, Z    +0.000, E1   -64.301, E3 +182112.792}
SPL {X  -160.000, Y  +670.465, Z    +0.000, E1   -64.283, E3 +182129.416}
SPL {X  -159.617, Y  +685.462, Z    +0.000, E1   -64.244, E3 +182145.143}
SPL {X  -158.001, Y  +699.614, Z    +0.000, E1   -64.013, E3 +182161.318}
SPL {X  -155.628, Y  +711.546, Z    +0.000, E1   -63.666, E3 +182175.987}
SPL {X  -152.846, Y  +721.708, Z    +0.000, E1   -63.251, E3 +182189.220}
SPL {X  -149.418, Y  +731.620, Z    +0.000, E1   -62.736, E3 +182202.775}
SPL {X  -145.585, Y  +740.770, Z    +0.000, E1   -62.119, E3 +182215.873}
SPL {X  -141.572, Y  +748.948, Z    +0.000, E1   -61.453, E3 +182227.998}
SPL {X  -137.548, Y  +756.134, Z    +0.000, E1   -60.743, E3 +182239.007}
SPL {X  -133.391, Y  +762.756, Z    +0.000, E1   -59.994, E3 +182249.324}
SPL {X  -109.419, Y  +791.137, Z    +0.000, E1   -49.920, E3 +182382.613}
ENDSPLINE

SPLINE
SPL {X  -148.079, Y  +735.002, Z    +0.000, E1   -35.426, E3 +182490.195}
SPL {X  -158.158, Y  +698.608, Z    +0.000, E1   -18.222, E3 +182502.848}
SPL {X  -159.870, Y  +680.839, Z    +0.000, E1    -6.577, E3 +182505.236}
SPL {X  -160.000, Y  +671.754, Z    +0.000, E1    +0.400, E3 +182505.595}
SPL {X  -160.000, Y  +663.703, Z    +0.000, E1   +12.763, E3 +182506.061}
SPL {X  -160.000, Y  +653.310, Z    +0.000, E1   +30.441, E3 +182507.531}
SPL {X  -160.000, Y  +640.945, Z    +0.000, E1   +44.811, E3 +182510.743}
SPL {X  -160.000, Y  +592.314, Z    +0.000, E1   +61.740, E3 +182532.736}
SPL {X  -160.000, Y  +478.009, Z    +0.000, E1   +65.091, E3 +182619.794}
SPL {X  -160.000, Y  +417.917, Z    +0.000, E1   +69.146, E3 +182639.964}
SPL {X  -160.000, Y  +403.867, Z    +0.000, E1   +68.803, E3 +182654.457}
SPL {X  -160.000, Y  +399.669, Z    +0.000, E1   +67.598, E3 +182668.328}
SPL {X  -160.000, Y  +392.628, Z    +0.000, E1   +66.554, E3 +182683.359}
SPL {X  -159.998, Y  +384.859, Z    +0.000, E1   +65.356, E3 +182700.287}
SPL {X  -159.712, Y  +376.098, Z    +0.000, E1   +64.333, E3 +182716.832}
SPL {X  -158.506, Y  +363.887, Z    +0.000, E1   +63.706, E3 +182734.224}
SPL {X  -155.923, Y  +349.812, Z    +0.000, E1   +63.321, E3 +182751.577}
SPL {X  -152.732, Y  +338.026, Z    +0.000, E1   +62.842, E3 +182767.112}
SPL {X  -149.257, Y  +328.060, Z    +0.000, E1   +62.292, E3 +182780.968}
SPL {X  -144.838, Y  +317.715, Z    +0.000, E1   +61.617, E3 +182795.974}
SPL {X  -139.661, Y  +307.631, Z    +0.000, E1   +60.727, E3 +182811.277}
SPL {X  -134.254, Y  +298.660, Z    +0.000, E1   +59.757, E3 +182825.325}
SPL {X  -111.782, Y  +271.224, Z    +0.000, E1   +50.030, E3 +182943.748}
ENDSPLINE

SPLINE
SPL {X  -142.230, Y  +312.416, Z    +0.000, E1   +39.081, E3 +183052.869}
SPL {X  -154.023, Y  +342.375, Z    +0.000, E1   +27.770, E3 +183069.326}
SPL {X  -159.227, Y  +369.989, Z    +0.000, E1   +12.792, E3 +183076.019}
SPL {X  -159.997, Y  +384.682, Z    +0.000, E1    +2.433, E3 +183077.383}
SPL {X  -160.000, Y  +388.025, Z    +0.000, E1    -0.434, E3 +183077.454}
SPL {X  -160.000, Y  +391.999, Z    +0.000, E1    -5.822, E3 +183077.599}
SPL {X  -160.000, Y  +397.968, Z    +0.000, E1   -15.492, E3 +183078.113}
SPL {X  -160.000, Y  +409.894, Z    +0.000, E1   -33.660, E3 +183080.220}
SPL {X  -160.000, Y  +457.050, Z    +0.000, E1   -59.500, E3 +183099.416}
SPL {X  -160.000, Y  +570.419, Z    +0.000, E1   -64.293, E3 +183184.981}
SPL {X  -160.000, Y  +587.690, Z    +0.000, E1   -64.299, E3 +183202.644}
SPL {X  -160.000, Y  +605.383, Z    +0.000, E1   -64.296, E3 +183220.742}
SPL {X  -160.000, Y  +621.010, Z    +0.000, E1   -64.279, E3 +183236.752}
SPL {X  -160.000, Y  +636.410, Z    +0.000, E1   -64.294, E3 +183252.481}
SPL {X  -160.000, Y  +654.238, Z    +0.000, E1   -64.301, E3 +183270.686}
SPL {X  -160.000, Y  +670.465, Z    +0.000, E1   -64.283, E3 +183287.310}
SPL {X  -159.617, Y  +685.462, Z    +0.000, E1   -64.244, E3 +183303.038}
SPL {X  -158.001, Y  +699.614, Z    +0.000, E1   -64.013, E3 +183319.213}
SPL {X  -155.628, Y  +711.546, Z    +0.000, E1   -63.666, E3 +183333.882}
SPL {X  -152.846, Y  +721.708, Z    +0.000, E1   -63.251, E3 +183347.115}
SPL {X  -149.418, Y  +731.620, Z    +0.000, E1   -62.736, E3 +183360.669}
SPL {X  -145.585, Y  +740.770, Z    +0.000, E1   -62.119, E3 +183373.768}
SPL {X  -141.572, Y  +748.948, Z    +0.000, E1   -61.453, E3 +183385.892}
SPL {X  -137.548, Y  +756.134, Z    +0.000, E1   -60.743, E3 +183396.901}
SPL {X  -133.391, Y  +762.756, Z    +0.000, E1   -59.994, E3 +183407.218}
SPL {X  -109.419, Y  +791.137, Z    +0.000, E1   -49.920, E3 +183540.507}
ENDSPLINE

SPLINE
SPL {X  -148.079, Y  +735.002, Z    +0.000, E1   -35.426, E3 +183648.090}
SPL {X  -158.158, Y  +698.608, Z    +0.000, E1   -18.222, E3 +183660.743}
SPL {X  -159.870, Y  +680.839, Z    +0.000, E1    -6.577, E3 +183663.131}
SPL {X  -160.000, Y  +671.754, Z    +0.000, E1    +0.400, E3 +183663.489}
SPL {X  -160.000, Y  +663.703, Z    +0.000, E1   +12.763, E3 +183663.955}
SPL {X  -160.000, Y  +653.310, Z    +0.000, E1   +30.441, E3 +183665.425}
SPL {X  -160.000, Y  +640.945, Z    +0.000, E1   +44.811, E3 +183668.637}
SPL {X  -160.000, Y  +592.314, Z    +0.000, E1   +61.740, E3 +183690.631}
SPL {X  -160.000, Y  +478.009, Z    +0.000, E1   +65.091, E3 +183777.689}
SPL {X  -160.000, Y  +417.917, Z    +0.000, E1   +69.146, E3 +183797.859}
SPL {X  -160.000, Y  +403.867, Z    +0.000, E1   +68.803, E3 +183812.351}
SPL {X  -160.000, Y  +399.669, Z    +0.000, E1   +67.598, E3 +183826.222}
SPL {X  -160.000, Y  +392.628, Z    +0.000, E1   +66.554, E3 +183841.253}
SPL {X  -159.998, Y  +384.859, Z    +0.000, E1   +65.356, E3 +183858.182}
SPL {X  -159.712, Y  +376.098, Z    +0.000, E1   +64.333, E3 +183874.726}
SPL {X  -158.506, Y  +363.887, Z    +0.000, E1   +63.706, E3 +183892.118}
SPL {X  -155.923, Y  +349.812, Z    +0.000, E1   +63.321, E3 +183909.471}
SPL {X  -152.732, Y  +338.026, Z    +0.000, E1   +62.842, E3 +183925.006}
SPL {X  -149.257, Y  +328.060, Z    +0.000, E1   +62.292, E3 +183938.863}
SPL {X  -144.838, Y  +317.715, Z    +0.000, E1   +61.617, E3 +183953.868}
SPL {X  -139.661, Y  +307.631, Z    +0.000, E1   +60.727, E3 +183969.172}
SPL {X  -134.254, Y  +298.660, Z    +0.000, E1   +59.757, E3 +183983.220}
SPL {X  -111.782, Y  +271.224, Z    +0.000, E1   +50.030, E3 +184101.643}
ENDSPLINE

SPLINE
SPL {X  -142.230, Y  +312.416, Z    +0.000, E1   +39.081, E3 +184210.763}
SPL {X  -154.023, Y  +342.375, Z    +0.000, E1   +27.770, E3 +184227.220}
SPL {X  -159.227, Y  +369.989, Z    +0.000, E1   +12.792, E3 +184233.913}
SPL {X  -159.997, Y  +384.682, Z    +0.000, E1    +2.433, E3 +184235.278}
SPL {X  -160.000, Y  +388.025, Z    +0.000, E1    -0.434, E3 +184235.348}
SPL {X  -160.000, Y  +391.999, Z    +0.000, E1    -5.822, E3 +184235.493}
SPL {X  -160.000, Y  +397.968, Z    +0.000, E1   -15.492, E3 +184236.007}
SPL {X  -160.000, Y  +409.894, Z    +0.000, E1   -33.660, E3 +184238.114}
SPL {X  -160.000, Y  +457.050, Z    +0.000, E1   -59.500, E3 +184257.311}
SPL {X  -160.000, Y  +570.419, Z    +0.000, E1   -64.293, E3 +184342.875}
SPL {X  -160.000, Y  +587.690, Z    +0.000, E1   -64.299, E3 +184360.538}
SPL {X  -160.000, Y  +605.383, Z    +0.000, E1   -64.296, E3 +184378.636}
SPL {X  -160.000, Y  +621.010, Z    +0.000, E1   -64.279, E3 +184394.646}
SPL {X  -160.000, Y  +636.410, Z    +0.000, E1   -64.294, E3 +184410.375}
SPL {X  -160.000, Y  +654.238, Z    +0.000, E1   -64.301, E3 +184428.581}
SPL {X  -160.000, Y  +670.465, Z    +0.000, E1   -64.283, E3 +184445.204}
SPL {X  -159.617, Y  +685.462, Z    +0.000, E1   -64.244, E3 +184460.932}
SPL {X  -158.001, Y  +699.614, Z    +0.000, E1   -64.013, E3 +184477.107}
SPL {X  -155.628, Y  +711.546, Z    +0.000, E1   -63.666, E3 +184491.776}
SPL {X  -152.846, Y  +721.708, Z    +0.000, E1   -63.251, E3 +184505.009}
SPL {X  -149.418, Y  +731.620, Z    +0.000, E1   -62.736, E3 +184518.563}
SPL {X  -145.585, Y  +740.770, Z    +0.000, E1   -62.119, E3 +184531.662}
SPL {X  -141.572, Y  +748.948, Z    +0.000, E1   -61.453, E3 +184543.786}
SPL {X  -137.548, Y  +756.134, Z    +0.000, E1   -60.743, E3 +184554.796}
SPL {X  -133.391, Y  +762.756, Z    +0.000, E1   -59.994, E3 +184565.112}
SPL {X  -109.419, Y  +791.137, Z    +0.000, E1   -49.920, E3 +184698.402}
ENDSPLINE

SPLINE
SPL {X  -148.079, Y  +735.002, Z    +0.000, E1   -35.426, E3 +184805.984}
SPL {X  -158.158, Y  +698.608, Z    +0.000, E1   -18.222, E3 +184818.637}
SPL {X  -159.870, Y  +680.839, Z    +0.000, E1    -6.577, E3 +184821.025}
SPL {X  -160.000, Y  +671.754, Z    +0.000, E1    +0.400, E3 +184821.383}
SPL {X  -160.000, Y  +663.703, Z    +0.000, E1   +12.763, E3 +184821.849}
SPL {X  -160.000, Y  +653.310, Z    +0.000, E1   +30.441, E3 +184823.319}
SPL {X  -160.000, Y  +640.945, Z    +0.000, E1   +44.811, E3 +184826.532}
SPL {X  -160.000, Y  +592.314, Z    +0.000, E1   +61.740, E3 +184848.525}
SPL {X  -160.000, Y  +478.009, Z    +0.000, E1   +65.091, E3 +184935.583}
SPL {X  -160.000, Y  +417.917, Z    +0.000, E1   +69.146, E3 +184955.753}
SPL {X  -160.000, Y  +403.867, Z    +0.000, E1   +68.803, E3 +184970.246}
SPL {X  -160.000, Y  +399.669, Z    +0.000, E1   +67.598, E3 +184984.117}
SPL {X  -160.000, Y  +392.628, Z    +0.000, E1   +66.554, E3 +184999.148}
SPL {X  -159.998, Y  +384.859, Z    +0.000, E1   +65.356, E3 +185016.076}
SPL {X  -159.712, Y  +376.098, Z    +0.000, E1   +64.333, E3 +185032.621}
SPL {X  -158.506, Y  +363.887, Z    +0.000, E1   +63.706, E3 +185050.012}
SPL {X  -155.923, Y  +349.812, Z    +0.000, E1   +63.321, E3 +185067.366}
SPL {X  -152.732, Y  +338.026, Z    +0.000, E1   +62.842, E3 +185082.900}
SPL {X  -149.257, Y  +328.060, Z    +0.000, E1   +62.292, E3 +185096.757}
SPL {X  -144.838, Y  +317.715, Z    +0.000, E1   +61.617, E3 +185111.763}
SPL {X  -139.661, Y  +307.631, Z    +0.000, E1   +60.727, E3 +185127.066}
SPL {X  -134.254, Y  +298.660, Z    +0.000, E1   +59.757, E3 +185141.114}
SPL {X  -111.782, Y  +271.224, Z    +0.000, E1   +50.030, E3 +185259.537}
ENDSPLINE

SPLINE
SPL {X  -142.230, Y  +312.416, Z    +0.000, E1   +39.081, E3 +185368.658}
SPL {X  -154.023, Y  +342.375, Z    +0.000, E1   +27.770, E3 +185385.114}
SPL {X  -159.227, Y  +369.989, Z    +0.000, E1   +12.792, E3 +185391.807}
SPL {X  -159.997, Y  +384.682, Z    +0.000, E1    +2.433, E3 +185393.172}
SPL {X  -160.000, Y  +388.025, Z    +0.000, E1    -0.434, E3 +185393.242}
SPL {X  -160.000, Y  +391.999, Z    +0.000, E1    -5.822, E3 +185393.387}
SPL {X  -160.000, Y  +397.968, Z    +0.000, E1   -15.492, E3 +185393.901}
SPL {X  -160.000, Y  +409.894, Z    +0.000, E1   -33.660, E3 +185396.009}
SPL {X  -160.000, Y  +457.050, Z    +0.000, E1   -59.500, E3 +185415.205}
SPL {X  -160.000, Y  +570.419, Z    +0.000, E1   -64.293, E3 +185500.770}
SPL {X  -160.000, Y  +587.690, Z    +0.000, E1   -64.299, E3 +185518.432}
SPL {X  -160.000, Y  +605.383, Z    +0.000, E1   -64.296, E3 +185536.531}
SPL {X  -160.000, Y  +621.010, Z    +0.000, E1   -64.279, E3 +185552.541}
SPL {X  -160.000, Y  +636.410, Z    +0.000, E1   -64.294, E3 +185568.270}
SPL {X  -160.000, Y  +654.238, Z    +0.000, E1   -64.301, E3 +185586.475}
SPL {X  -160.000, Y  +670.465, Z    +0.000, E1   -64.283, E3 +185603.099}
SPL {X  -159.617, Y  +685.462, Z    +0.000, E1   -64.244, E3 +185618.826}
SPL {X  -158.001, Y  +699.614, Z    +0.000, E1   -64.013, E3 +185635.001}
SPL {X  -155.628, Y  +711.546, Z    +0.000, E1   -63.666, E3 +185649.670}
SPL {X  -152.846, Y  +721.708, Z    +0.000, E1   -63.251, E3 +185662.903}
SPL {X  -149.418, Y  +731.620, Z    +0.000, E1   -62.736, E3 +185676.458}
SPL {X  -145.585, Y  +740.770, Z    +0.000, E1   -62.119, E3 +185689.556}
SPL {X  -141.572, Y  +748.948, Z    +0.000, E1   -61.453, E3 +185701.681}
SPL {X  -137.548, Y  +756.134, Z    +0.000, E1   -60.743, E3 +185712.690}
SPL {X  -133.391, Y  +762.756, Z    +0.000, E1   -59.994, E3 +185723.007}
SPL {X  -109.419, Y  +791.137, Z    +0.000, E1   -49.920, E3 +185856.296}
ENDSPLINE

SPLINE
SPL {X  -148.079, Y  +735.002, Z    +0.000, E1   -35.426, E3 +185963.878}
SPL {X  -158.158, Y  +698.608, Z    +0.000, E1   -18.222, E3 +185976.531}
SPL {X  -159.870, Y  +680.839, Z    +0.000, E1    -6.577, E3 +185978.919}
SPL {X  -160.000, Y  +671.754, Z    +0.000, E1    +0.400, E3 +185979.278}
SPL {X  -160.000, Y  +663.703, Z    +0.000, E1   +12.763, E3 +185979.744}
SPL {X  -160.000, Y  +653.310, Z    +0.000, E1   +30.441, E3 +185981.214}
SPL {X  -160.000, Y  +640.945, Z    +0.000, E1   +44.811, E3 +185984.426}
SPL {X  -160.000, Y  +592.314, Z    +0.000, E1   +61.740, E3 +186006.419}
SPL {X  -160.000, Y  +478.009, Z    +0.000, E1   +65.091, E3 +186093.477}
SPL {X  -160.000, Y  +417.917, Z    +0.000, E1   +69.146, E3 +186113.647}
SPL {X  -160.000, Y  +403.867, Z    +0.000, E1   +68.803, E3 +186128.140}
SPL {X  -160.000, Y  +399.669, Z    +0.000, E1   +67.598, E3 +186142.011}
SPL {X  -160.000, Y  +392.628, Z    +0.000, E1   +66.554, E3 +186157.042}
SPL {X  -159.998, Y  +384.859, Z    +0.000, E1   +65.356, E3 +186173.970}
SPL {X  -159.712, Y  +376.098, Z    +0.000, E1   +64.333, E3 +186190.515}
SPL {X  -158.506, Y  +363.887, Z    +0.000, E1   +63.706, E3 +186207.907}
SPL {X  -155.923, Y  +349.812, Z    +0.000, E1   +63.321, E3 +186225.260}
SPL {X  -152.732, Y  +338.026, Z    +0.000, E1   +62.842, E3 +186240.795}
SPL {X  -149.257, Y  +328.060, Z    +0.000, E1   +62.292, E3 +186254.651}
SPL {X  -144.838, Y  +317.715, Z    +0.000, E1   +61.617, E3 +186269.657}
SPL {X  -139.661, Y  +307.631, Z    +0.000, E1   +60.727, E3 +186284.960}
SPL {X  -134.254, Y  +298.660, Z    +0.000, E1   +59.757, E3 +186299.008}
SPL {X  -111.782, Y  +271.224, Z    +0.000, E1   +50.030, E3 +186417.431}
ENDSPLINE

SPLINE
SPL {X  -142.230, Y  +312.416, Z    +0.000, E1   +39.081, E3 +186526.552}
SPL {X  -154.023, Y  +342.375, Z    +0.000, E1   +27.770, E3 +186543.009}
SPL {X  -159.227, Y  +369.989, Z    +0.000, E1   +12.792, E3 +186549.702}
SPL {X  -159.997, Y  +384.682, Z    +0.000, E1    +2.433, E3 +186551.066}
SPL {X  -160.000, Y  +388.025, Z    +0.000, E1    -0.434, E3 +186551.137}
SPL {X  -160.000, Y  +391.999, Z    +0.000, E1    -5.822, E3 +186551.281}
SPL {X  -160.000, Y  +397.968, Z    +0.000, E1   -15.492, E3 +186551.796}
SPL {X  -160.000, Y  +409.894, Z    +0.000, E1   -33.660, E3 +186553.903}
SPL {X  -160.000, Y  +457.050, Z    +0.000, E1   -59.500, E3 +186573.099}
SPL {X  -160.000, Y  +570.419, Z    +0.000, E1   -64.293, E3 +186658.664}
SPL {X  -160.000, Y  +587.690, Z    +0.000, E1   -64.299, E3 +186676.327}
SPL {X  -160.000, Y  +605.383, Z    +0.000, E1   -64.296, E3 +186694.425}
SPL {X  -160.000, Y  +621.010, Z    +0.000, E1   -64.279, E3 +186710.435}
SPL {X  -160.000, Y  +636.410, Z    +0.000, E1   -64.294, E3 +186726.164}
SPL {X  -160.000, Y  +654.238, Z    +0.000, E1   -64.301, E3 +186744.369}
SPL {X  -160.000, Y  +670.465, Z    +0.000, E1   -64.283, E3 +186760.993}
SPL {X  -159.617, Y  +685.462, Z    +0.000, E1   -64.244, E3 +186776.721}
SPL {X  -158.001, Y  +699.614, Z    +0.000, E1   -64.013, E3 +186792.896}
SPL {X  -155.628, Y  +711.546, Z    +0.000, E1   -63.666, E3 +186807.565}
SPL {X  -152.846, Y  +721.708, Z    +0.000, E1   -63.251, E3 +186820.798}
SPL {X  -149.418, Y  +731.620, Z    +0.000, E1   -62.736, E3 +186834.352}
SPL {X  -145.585, Y  +740.770, Z    +0.000, E1   -62.119, E3 +186847.451}
SPL {X  -141.572, Y  +748.948, Z    +0.000, E1   -61.453, E3 +186859.575}
SPL {X  -137.548, Y  +756.134, Z    +0.000, E1   -60.743, E3 +186870.584}
SPL {X  -133.391, Y  +762.756, Z    +0.000, E1   -59.994, E3 +186880.901}
SPL {X  -109.419, Y  +791.137, Z    +0.000, E1   -49.920, E3 +187014.190}
ENDSPLINE

SPLINE
SPL {X  -148.079, Y  +735.002, Z    +0.000, E1   -35.426, E3 +187121.773}
SPL {X  -158.158, Y  +698.608, Z    +0.000, E1   -18.222, E3 +187134.426}
SPL {X  -159.870, Y  +680.839, Z    +0.000, E1    -6.577, E3 +187136.814}
SPL {X  -160.000, Y  +671.754, Z    +0.000, E1    +0.400, E3 +187137.172}
SPL {X  -160.000, Y  +663.703, Z    +0.000, E1   +12.763, E3 +187137.638}
SPL {X  -160.000, Y  +653.310, Z    +0.000, E1   +30.441, E3 +187139.108}
SPL {X  -160.000, Y  +640.945, Z    +0.000, E1   +44.811, E3 +187142.320}
SPL {X  -160.000, Y  +592.314, Z    +0.000, E1   +61.740, E3 +187164.314}
SPL {X  -160.000, Y  +478.009, Z    +0.000, E1   +65.091, E3 +187251.372}
SPL {X  -160.000, Y  +417.917, Z    +0.000, E1   +69.146, E3 +187271.542}
SPL {X  -160.000, Y  +403.867, Z    +0.000, E1   +68.803, E3 +187286.034}
SPL {X  -160.000, Y  +399.669, Z    +0.000, E1   +67.598, E3 +187299.905}
SPL {X  -160.000, Y  +392.628, Z    +0.000, E1   +66.554, E3 +187314.936}
SPL {X  -159.998, Y  +384.859, Z    +0.000, E1   +65.356, E3 +187331.865}
SPL {X  -159.712, Y  +376.098, Z    +0.000, E1   +64.333, E3 +187348.409}
SPL {X  -158.506, Y  +363.887, Z    +0.000, E1   +63.706, E3 +187365.801}
SPL {X  -155.923, Y  +349.812, Z    +0.000, E1   +63.321, E3 +187383.154}
SPL {X  -152.732, Y  +338.026, Z    +0.000, E1   +62.842, E3 +187398.689}
SPL {X  -149.257, Y  +328.060, Z    +0.000, E1   +62.292, E3 +187412.545}
SPL {X  -144.838, Y  +317.715, Z    +0.000, E1   +61.617, E3 +187427.551}
SPL {X  -139.661, Y  +307.631, Z    +0.000, E1   +60.727, E3 +187442.855}
SPL {X  -134.254, Y  +298.660, Z    +0.000, E1   +59.757, E3 +187456.903}
SPL {X  -111.782, Y  +271.224, Z    +0.000, E1   +50.030, E3 +187575.326}
ENDSPLINE

SPLINE
SPL {X  -142.230, Y  +312.416, Z    +0.000, E1   +39.081, E3 +187684.446}
SPL {X  -154.023, Y  +342.375, Z    +0.000, E1   +27.770, E3 +187700.903}
SPL {X  -159.227, Y  +369.989, Z    +0.000, E1   +12.792, E3 +187707.596}
SPL {X  -159.997, Y  +384.682, Z    +0.000, E1    +2.433, E3 +187708.961}
SPL {X  -160.000, Y  +388.025, Z    +0.000, E1    -0.434, E3 +187709.031}
SPL {X  -160.000, Y  +391.999, Z    +0.000, E1    -5.822, E3 +187709.176}
SPL {X  -160.000, Y  +397.968, Z    +0.000, E1   -15.492, E3 +187709.690}
SPL {X  -160.000, Y  +409.894, Z    +0.000, E1   -33.660, E3 +187711.797}
SPL {X  -160.000, Y  +457.050, Z    +0.000, E1   -59.500, E3 +187730.994}
SPL {X  -160.000, Y  +570.419, Z    +0.000, E1   -64.293, E3 +187816.558}
SPL {X  -160.000, Y  +587.690, Z    +0.000, E1   -64.299, E3 +187834.221}
SPL {X  -160.000, Y  +605.383, Z    +0.000, E1   -64.296, E3 +187852.319}
SPL {X  -160.000, Y  +621.010, Z    +0.000, E1   -64.279, E3 +187868.329}
SPL {X  -160.000, Y  +636.410, Z    +0.000, E1   -64.294, E3 +187884.058}
SPL {X  -160.000, Y  +654.238, Z    +0.000, E1   -64.301, E3 +187902.264}
SPL {X  -160.000, Y  +670.465, Z    +0.000, E1   -64.283, E3 +187918.887}
SPL {X  -159.617, Y  +685.462, Z    +0.000, E1   -64.244, E3 +187934.615}
SPL {X  -158.001, Y  +699.614, Z    +0.000, E1   -64.013, E3 +187950.790}
SPL {X  -155.628, Y  +711.546, Z    +0.000, E1   -63.666, E3 +187965.459}
SPL {X  -152.846, Y  +721.708, Z    +0.000, E1   -63.251, E3 +187978.692}
SPL {X  -149.418, Y  +731.620, Z    +0.000, E1   -62.736, E3 +187992.246}
SPL {X  -145.585, Y  +740.770, Z    +0.000, E1   -62.119, E3 +188005.345}
SPL {X  -141.572, Y  +748.948, Z    +0.000, E1   -61.453, E3 +188017.469}
SPL {X  -137.548, Y  +756.134, Z    +0.000, E1   -60.743, E3 +188028.479}
SPL {X  -133.391, Y  +762.756, Z    +0.000, E1   -59.994, E3 +188038.795}
SPL {X  -109.419, Y  +791.137, Z    +0.000, E1   -49.920, E3 +188172.085}
ENDSPLINE

SPLINE
SPL {X  -148.079, Y  +735.002, Z    +0.000, E1   -35.426, E3 +188279.667}
SPL {X  -158.158, Y  +698.608, Z    +0.000, E1   -18.222, E3 +188292.320}
SPL {X  -159.870, Y  +680.839, Z    +0.000, E1    -6.577, E3 +188294.708}
SPL {X  -160.000, Y  +671.754, Z    +0.000, E1    +0.400, E3 +188295.066}
SPL {X  -160.000, Y  +663.703, Z    +0.000, E1   +12.763, E3 +188295.532}
SPL {X  -160.000, Y  +653.310, Z    +0.000, E1   +30.441, E3 +188297.002}
SPL {X  -160.000, Y  +640.945, Z    +0.000, E1   +44.811, E3 +188300.215}
SPL {X  -160.000, Y  +592.314, Z    +0.000, E1   +61.740, E3 +188322.208}
SPL {X  -160.000, Y  +478.009, Z    +0.000, E1   +65.091, E3 +188409.266}
SPL {X  -160.000, Y  +417.917, Z    +0.000, E1   +69.146, E3 +188429.436}
SPL {X  -160.000, Y  +403.867, Z    +0.000, E1   +68.803, E3 +188443.929}
SPL {X  -160.000, Y  +399.669, Z    +0.000, E1   +67.598, E3 +188457.800}
SPL {X  -160.000, Y  +392.628, Z    +0.000, E1   +66.554, E3 +188472.831}
SPL {X  -159.998, Y  +384.859, Z    +0.000, E1   +65.356, E3 +188489.759}
SPL {X  -159.712, Y  +376.098, Z    +0.000, E1   +64.333, E3 +188506.303}
SPL {X  -158.506, Y  +363.887, Z    +0.000, E1   +63.706, E3 +188523.695}
SPL {X  -155.923, Y  +349.812, Z    +0.000, E1   +63.321, E3 +188541.049}
SPL {X  -152.732, Y  +338.026, Z    +0.000, E1   +62.842, E3 +188556.583}
SPL {X  -149.257, Y  +328.060, Z    +0.000, E1   +62.292, E3 +188570.440}
SPL {X  -144.838, Y  +317.715, Z    +0.000, E1   +61.617, E3 +188585.446}
SPL {X  -139.661, Y  +307.631, Z    +0.000, E1   +60.727, E3 +188600.749}
SPL {X  -134.254, Y  +298.660, Z    +0.000, E1   +59.757, E3 +188614.797}
SPL {X  -111.782, Y  +271.224, Z    +0.000, E1   +50.030, E3 +188733.220}
ENDSPLINE

SPLINE
SPL {X  -142.230, Y  +312.416, Z    +0.000, E1   +39.081, E3 +188842.341}
SPL {X  -154.023, Y  +342.375, Z    +0.000, E1   +27.770, E3 +188858.797}
SPL {X  -159.227, Y  +369.989, Z    +0.000, E1   +12.792, E3 +188865.490}
SPL {X  -159.997, Y  +384.682, Z    +0.000, E1    +2.433, E3 +188866.855}
SPL {X  -160.000, Y  +388.025, Z    +0.000, E1    -0.434, E3 +188866.925}
SPL {X  -160.000, Y  +391.999, Z    +0.000, E1    -5.822, E3 +188867.070}
SPL {X  -160.000, Y  +397.968, Z    +0.000, E1   -15.492, E3 +188867.584}
SPL {X  -160.000, Y  +409.894, Z    +0.000, E1   -33.660, E3 +188869.692}
SPL {X  -160.000, Y  +457.050, Z    +0.000, E1   -59.500, E3 +188888.888}
SPL {X  -160.000, Y  +570.419, Z    +0.000, E1   -64.293, E3 +188974.453}
SPL {X  -160.000, Y  +587.690, Z    +0.000, E1   -64.299, E3 +188992.115}
SPL {X  -160.000, Y  +605.383, Z    +0.000, E1   -64.296, E3 +189010.214}
SPL {X  -160.000, Y  +621.010, Z    +0.000, E1   -64.279, E3 +189026.224}
SPL {X  -160.000, Y  +636.410, Z    +0.000, E1   -64.294, E3 +189041.953}
SPL {X  -160.000, Y  +654.238, Z    +0.000, E1   -64.301, E3 +189060.158}
SPL {X  -160.000, Y  +670.465, Z    +0.000, E1   -64.283, E3 +189076.782}
SPL {X  -159.617, Y  +685.462, Z    +0.000, E1   -64.244, E3 +189092.509}
SPL {X  -158.001, Y  +699.614, Z    +0.000, E1   -64.013, E3 +189108.684}
SPL {X  -155.628, Y  +711.546, Z    +0.000, E1   -63.666, E3 +189123.353}
SPL {X  -152.846, Y  +721.708, Z    +0.000, E1   -63.251, E3 +189136.586}
SPL {X  -149.418, Y  +731.620, Z    +0.000, E1   -62.736, E3 +189150.141}
SPL {X  -145.585, Y  +740.770, Z    +0.000, E1   -62.119, E3 +189163.239}
SPL {X  -141.572, Y  +748.948, Z    +0.000, E1   -61.453, E3 +189175.364}
SPL {X  -137.548, Y  +756.134, Z    +0.000, E1   -60.743, E3 +189186.373}
SPL {X  -133.391, Y  +762.756, Z    +0.000, E1   -59.994, E3 +189196.690}
SPL {X  -109.419, Y  +791.137, Z    +0.000, E1   -49.920, E3 +189329.979}
ENDSPLINE

SPLINE
SPL {X  -148.079, Y  +735.002, Z    +0.000, E1   -35.426, E3 +189437.561}
SPL {X  -158.158, Y  +698.608, Z    +0.000, E1   -18.222, E3 +189450.214}
SPL {X  -159.870, Y  +680.839, Z    +0.000, E1    -6.577, E3 +189452.602}
SPL {X  -160.000, Y  +671.754, Z    +0.000, E1    +0.400, E3 +189452.961}
SPL {X  -160.000, Y  +663.703, Z    +0.000, E1   +12.763, E3 +189453.426}
SPL {X  -160.000, Y  +653.310, Z    +0.000, E1   +30.441, E3 +189454.897}
SPL {X  -160.000, Y  +640.945, Z    +0.000, E1   +44.811, E3 +189458.109}
SPL {X  -160.000, Y  +592.314, Z    +0.000, E1   +61.740, E3 +189480.102}
SPL {X  -160.000, Y  +478.009, Z    +0.000, E1   +65.091, E3 +189567.160}
SPL {X  -160.000, Y  +417.917, Z    +0.000, E1   +69.146, E3 +189587.330}
SPL {X  -160.000, Y  +403.867, Z    +0.000, E1   +68.803, E3 +189601.823}
SPL {X  -160.000, Y  +399.669, Z    +0.000, E1   +67.598, E3 +189615.694}
SPL {X  -160.000, Y  +392.628, Z    +0.000, E1   +66.554, E3 +189630.725}
SPL {X  -159.998, Y  +384.859, Z    +0.000, E1   +65.356, E3 +189647.653}
SPL {X  -159.712, Y  +376.098, Z    +0.000, E1   +64.333, E3 +189664.198}
SPL {X  -158.506, Y  +363.887, Z    +0.000, E1   +63.706, E3 +189681.590}
SPL {X  -155.923, Y  +349.812, Z    +0.000, E1   +63.321, E3 +189698.943}
SPL {X  -152.732, Y  +338.026, Z    +0.000, E1   +62.842, E3 +189714.478}
SPL {X  -149.257, Y  +328.060, Z    +0.000, E1   +62.292, E3 +189728.334}
SPL {X  -144.838, Y  +317.715, Z    +0.000, E1   +61.617, E3 +189743.340}
SPL {X  -139.661, Y  +307.631, Z    +0.000, E1   +60.727, E3 +189758.643}
SPL {X  -134.254, Y  +298.660, Z    +0.000, E1   +59.757, E3 +189772.691}
SPL {X  -111.782, Y  +271.224, Z    +0.000, E1   +50.030, E3 +189891.114}
ENDSPLINE

SPLINE
SPL {X  -142.230, Y  +312.416, Z    +0.000, E1   +39.081, E3 +190000.235}
SPL {X  -154.023, Y  +342.375, Z    +0.000, E1   +27.770, E3 +190016.692}
SPL {X  -159.227, Y  +369.989, Z    +0.000, E1   +12.792, E3 +190023.385}
SPL {X  -159.997, Y  +384.682, Z    +0.000, E1    +2.433, E3 +190024.749}
SPL {X  -160.000, Y  +388.025, Z    +0.000, E1    -0.434, E3 +190024.820}
SPL {X  -160.000, Y  +391.999, Z    +0.000, E1    -5.822, E3 +190024.964}
SPL {X  -160.000, Y  +397.968, Z    +0.000, E1   -15.492, E3 +190025.479}
SPL {X  -160.000, Y  +409.894, Z    +0.000, E1   -33.660, E3 +190027.586}
SPL {X  -160.000, Y  +457.050, Z    +0.000, E1   -59.500, E3 +190046.782}
SPL {X  -160.000, Y  +570.419, Z    +0.000, E1   -64.293, E3 +190132.347}
SPL {X  -160.000, Y  +587.690, Z    +0.000, E1   -64.299, E3 +190150.010}
SPL {X  -160.000, Y  +605.383, Z    +0.000, E1   -64.296, E3 +190168.108}
SPL {X  -160.000, Y  +621.010, Z    +0.000, E1   -64.279, E3 +190184.118}
SPL {X  -160.000, Y  +636.410, Z    +0.000, E1   -64.294, E3 +190199.847}
SPL {X  -160.000, Y  +654.238, Z    +0.000, E1   -64.301, E3 +190218.052}
SPL {X  -160.000, Y  +670.465, Z    +0.000, E1   -64.283, E3 +190234.676}
SPL {X  -159.617, Y  +685.462, Z    +0.000, E1   -64.244, E3 +190250.404}
SPL {X  -158.001, Y  +699.614, Z    +0.000, E1   -64.013, E3 +190266.579}
SPL {X  -155.628, Y  +711.546, Z    +0.000, E1   -63.666, E3 +190281.248}
SPL {X  -152.846, Y  +721.708, Z    +0.000, E1   -63.251, E3 +190294.480}
SPL {X  -149.418, Y  +731.620, Z    +0.000, E1   -62.736, E3 +190308.035}
SPL {X  -145.585, Y  +740.770, Z    +0.000, E1   -62.119, E3 +190321.134}
SPL {X  -141.572, Y  +748.948, Z    +0.000, E1   -61.453, E3 +190333.258}
SPL {X  -137.548, Y  +756.134, Z    +0.000, E1   -60.743, E3 +190344.267}
SPL {X  -133.391, Y  +762.756, Z    +0.000, E1   -59.994, E3 +190354.584}
SPL {X  -109.419, Y  +791.137, Z    +0.000, E1   -49.920, E3 +190487.873}
ENDSPLINE

SPLINE
SPL {X  -148.079, Y  +735.002, Z    +0.000, E1   -35.426, E3 +190595.456}
SPL {X  -158.158, Y  +698.608, Z    +0.000, E1   -18.222, E3 +190608.109}
SPL {X  -159.870, Y  +680.839, Z    +0.000, E1    -6.577, E3 +190610.496}
SPL {X  -160.000, Y  +671.754, Z    +0.000, E1    +0.400, E3 +190610.855}
SPL {X  -160.000, Y  +663.703, Z    +0.000, E1   +12.763, E3 +190611.321}
SPL {X  -160.000, Y  +653.310, Z    +0.000, E1   +30.441, E3 +190612.791}
SPL {X  -160.000, Y  +640.945, Z    +0.000, E1   +44.811, E3 +190616.003}
SPL {X  -160.000, Y  +592.314, Z    +0.000, E1   +61.740, E3 +190637.997}
SPL {X  -160.000, Y  +478.009, Z    +0.000, E1   +65.091, E3 +190725.055}
SPL {X  -160.000, Y  +417.917, Z    +0.000, E1   +69.146, E3 +190745.225}
SPL {X  -160.000, Y  +403.867, Z    +0.000, E1   +68.803, E3 +190759.717}
SPL {X  -160.000, Y  +399.669, Z    +0.000, E1   +67.598, E3 +190773.588}
SPL {X  -160.000, Y  +392.628, Z    +0.000, E1   +66.554, E3 +190788.619}
SPL {X  -159.998, Y  +384.859, Z    +0.000, E1   +65.356, E3 +190805.548}
SPL {X  -159.712, Y  +376.098, Z    +0.000, E1   +64.333, E3 +190822.092}
SPL {X  -158.506, Y  +363.887, Z    +0.000, E1   +63.706, E3 +190839.484}
SPL {X  -155.923, Y  +349.812, Z    +0.000, E1   +63.321, E3 +190856.837}
SPL {X  -152.732, Y  +338.026, Z    +0.000, E1   +62.842, E3 +190872.372}
SPL {X  -149.257, Y  +328.060, Z    +0.000, E1   +62.292, E3 +190886.228}
SPL {X  -144.838, Y  +317.715, Z    +0.000, E1   +61.617, E3 +190901.234}
SPL {X  -139.661, Y  +307.631, Z    +0.000, E1   +60.727, E3 +190916.538}
SPL {X  -134.254, Y  +298.660, Z    +0.000, E1   +59.757, E3 +190930.586}
SPL {X  -111.782, Y  +271.224, Z    +0.000, E1   +50.030, E3 +191049.009}
ENDSPLINE

SPLINE
SPL {X  -142.230, Y  +312.416, Z    +0.000, E1   +39.081, E3 +191158.129}
SPL {X  -154.023, Y  +342.375, Z    +0.000, E1   +27.770, E3 +191174.586}
SPL {X  -159.227, Y  +369.989, Z    +0.000, E1   +12.792, E3 +191181.279}
SPL {X  -159.997, Y  +384.682, Z    +0.000, E1    +2.433, E3 +191182.644}
SPL {X  -160.000, Y  +388.025, Z    +0.000, E1    -0.434, E3 +191182.714}
SPL {X  -160.000, Y  +391.999, Z    +0.000, E1    -5.822, E3 +191182.859}
SPL {X  -160.000, Y  +397.968, Z    +0.000, E1   -15.492, E3 +191183.373}
SPL {X  -160.000, Y  +409.894, Z    +0.000, E1   -33.660, E3 +191185.480}
SPL {X  -160.000, Y  +457.050, Z    +0.000, E1   -59.500, E3 +191204.677}
SPL {X  -160.000, Y  +570.419, Z    +0.000, E1   -64.293, E3 +191290.241}
SPL {X  -160.000, Y  +587.690, Z    +0.000, E1   -64.299, E3 +191307.904}
SPL {X  -160.000, Y  +605.383, Z    +0.000, E1   -64.296, E3 +191326.002}
SPL {X  -160.000, Y  +621.010, Z    +0.000, E1   -64.279, E3 +191342.012}
SPL {X  -160.000, Y  +636.410, Z    +0.000, E1   -64.294, E3 +191357.741}
SPL {X  -160.000, Y  +654.238, Z    +0.000, E1   -64.301, E3 +191375.947}
SPL {X  -160.000, Y  +670.465, Z    +0.000, E1   -64.283, E3 +191392.570}
SPL {X  -159.617, Y  +685.462, Z    +0.000, E1   -64.244, E3 +191408.298}
SPL {X  -158.001, Y  +699.614, Z    +0.000, E1   -64.013, E3 +191424.473}
SPL {X  -155.628, Y  +711.546, Z    +0.000, E1   -63.666, E3 +191439.142}
SPL {X  -152.846, Y  +721.708, Z    +0.000, E1   -63.251, E3 +191452.375}
SPL {X  -149.418, Y  +731.620, Z    +0.000, E1   -62.736, E3 +191465.929}
SPL {X  -145.585, Y  +740.770, Z    +0.000, E1   -62.119, E3 +191479.028}
SPL {X  -141.572, Y  +748.948, Z    +0.000, E1   -61.453, E3 +191491.152}
SPL {X  -137.548, Y  +756.134, Z    +0.000, E1   -60.743, E3 +191502.162}
SPL {X  -133.391, Y  +762.756, Z    +0.000, E1   -59.994, E3 +191512.478}
SPL {X  -109.419, Y  +791.137, Z    +0.000, E1   -49.920, E3 +191645.767}
ENDSPLINE

SPLINE
SPL {X  -148.079, Y  +735.002, Z    +0.000, E1   -35.426, E3 +191753.350}
SPL {X  -158.158, Y  +698.608, Z    +0.000, E1   -18.222, E3 +191766.003}
SPL {X  -159.870, Y  +680.839, Z    +0.000, E1    -6.577, E3 +191768.391}
SPL {X  -160.000, Y  +671.754, Z    +0.000, E1    +0.400, E3 +191768.749}
SPL {X  -160.000, Y  +663.703, Z    +0.000, E1   +12.763, E3 +191769.215}
SPL {X  -160.000, Y  +653.310, Z    +0.000, E1   +30.441, E3 +191770.685}
SPL {X  -160.000, Y  +640.945, Z    +0.000, E1   +44.811, E3 +191773.897}
SPL {X  -160.000, Y  +592.314, Z    +0.000, E1   +61.740, E3 +191795.891}
SPL {X  -160.000, Y  +478.009, Z    +0.000, E1   +65.091, E3 +191882.949}
SPL {X  -160.000, Y  +417.917, Z    +0.000, E1   +69.146, E3 +191903.119}
SPL {X  -160.000, Y  +403.867, Z    +0.000, E1   +68.803, E3 +191917.612}
SPL {X  -160.000, Y  +399.669, Z    +0.000, E1   +67.598, E3 +191931.483}
SPL {X  -160.000, Y  +392.628, Z    +0.000, E1   +66.554, E3 +191946.514}
SPL {X  -159.998, Y  +384.859, Z    +0.000, E1   +65.356, E3 +191963.442}
SPL {X  -159.712, Y  +376.098, Z    +0.000, E1   +64.333, E3 +191979.986}
SPL {X  -158.506, Y  +363.887, Z    +0.000, E1   +63.706, E3 +191997.378}
SPL {X  -155.923, Y  +349.812, Z    +0.000, E1   +63.321, E3 +192014.732}
SPL {X  -152.732, Y  +338.026, Z    +0.000, E1   +62.842, E3 +192030.266}
SPL {X  -149.257, Y  +328.060, Z    +0.000, E1   +62.292, E3 +192044.123}
SPL {X  -144.838, Y  +317.715, Z    +0.000, E1   +61.617, E3 +192059.129}
SPL {X  -139.661, Y  +307.631, Z    +0.000, E1   +60.727, E3 +192074.432}
SPL {X  -134.254, Y  +298.660, Z    +0.000, E1   +59.757, E3 +192088.480}
SPL {X  -111.782, Y  +271.224, Z    +0.000, E1   +50.030, E3 +192206.903}
ENDSPLINE

SPLINE
SPL {X  -142.230, Y  +312.416, Z    +0.000, E1   +39.081, E3 +192316.023}
SPL {X  -154.023, Y  +342.375, Z    +0.000, E1   +27.770, E3 +192332.480}
SPL {X  -159.227, Y  +369.989, Z    +0.000, E1   +12.792, E3 +192339.173}
SPL {X  -159.997, Y  +384.682, Z    +0.000, E1    +2.433, E3 +192340.538}
SPL {X  -160.000, Y  +388.025, Z    +0.000, E1    -0.434, E3 +192340.608}
SPL {X  -160.000, Y  +391.999, Z    +0.000, E1    -5.822, E3 +192340.753}
SPL {X  -160.000, Y  +397.968, Z    +0.000, E1   -15.492, E3 +192341.267}
SPL {X  -160.000, Y  +409.894, Z    +0.000, E1   -33.660, E3 +192343.374}
SPL {X  -160.000, Y  +457.050, Z    +0.000, E1   -59.500, E3 +192362.571}
SPL {X  -160.000, Y  +570.419, Z    +0.000, E1   -64.293, E3 +192448.136}
SPL {X  -160.000, Y  +587.690, Z    +0.000, E1   -64.299, E3 +192465.798}
SPL {X  -160.000, Y  +605.383, Z    +0.000, E1   -64.296, E3 +192483.897}
SPL {X  -160.000, Y  +621.010, Z    +0.000, E1   -64.279, E3 +192499.907}
SPL {X  -160.000, Y  +636.410, Z    +0.000, E1   -64.294, E3 +192515.635}
SPL {X  -160.000, Y  +654.238, Z    +0.000, E1   -64.301, E3 +192533.841}
SPL {X  -160.000, Y  +670.465, Z    +0.000, E1   -64.283, E3 +192550.464}
SPL {X  -159.617, Y  +685.462, Z    +0.000, E1   -64.244, E3 +192566.192}
SPL {X  -158.001, Y  +699.614, Z    +0.000, E1   -64.013, E3 +192582.367}
SPL {X  -155.628, Y  +711.546, Z    +0.000, E1   -63.666, E3 +192597.036}
SPL {X  -152.846, Y  +721.708, Z    +0.000, E1   -63.251, E3 +192610.269}
SPL {X  -149.418, Y  +731.620, Z    +0.000, E1   -62.736, E3 +192623.824}
SPL {X  -145.585, Y  +740.770, Z    +0.000, E1   -62.119, E3 +192636.922}
SPL {X  -141.572, Y  +748.948, Z    +0.000, E1   -61.453, E3 +192649.046}
SPL {X  -137.548, Y  +756.134, Z    +0.000, E1   -60.743, E3 +192660.056}
SPL {X  -133.391, Y  +762.756, Z    +0.000, E1   -59.994, E3 +192670.373}
SPL {X  -109.419, Y  +791.137, Z    +0.000, E1   -49.920, E3 +192803.662}
ENDSPLINE

SPLINE
SPL {X  -148.079, Y  +735.002, Z    +0.000, E1   -35.426, E3 +192911.244}
SPL {X  -158.158, Y  +698.608, Z    +0.000, E1   -18.222, E3 +192923.897}
SPL {X  -159.870, Y  +680.839, Z    +0.000, E1    -6.577, E3 +192926.285}
SPL {X  -160.000, Y  +671.754, Z    +0.000, E1    +0.400, E3 +192926.644}
SPL {X  -160.000, Y  +663.703, Z    +0.000, E1   +12.763, E3 +192927.109}
SPL {X  -160.000, Y  +653.310, Z    +0.000, E1   +30.441, E3 +192928.580}
SPL {X  -160.000, Y  +640.945, Z    +0.000, E1   +44.811, E3 +192931.792}
SPL {X  -160.000, Y  +592.314, Z    +0.000, E1   +61.740, E3 +192953.785}
SPL {X  -160.000, Y  +478.009, Z    +0.000, E1   +65.091, E3 +193040.843}
SPL {X  -160.000, Y  +417.917, Z    +0.000, E1   +69.146, E3 +193061.013}
SPL {X  -160.000, Y  +403.867, Z    +0.000, E1   +68.803, E3 +193075.506}
SPL {X  -160.000, Y  +399.669, Z    +0.000, E1   +67.598, E3 +193089.377}
SPL {X  -160.000, Y  +392.628, Z    +0.000, E1   +66.554, E3 +193104.408}
SPL {X  -159.998, Y  +384.859, Z    +0.000, E1   +65.356, E3 +193121.336}
SPL {X  -159.712, Y  +376.098, Z    +0.000, E1   +64.333, E3 +193137.881}
SPL {X  -158.506, Y  +363.887, Z    +0.000, E1   +63.706, E3 +193155.273}
SPL {X  -155.923, Y  +349.812, Z    +0.000, E1   +63.321, E3 +193172.626}
SPL {X  -152.732, Y  +338.026, Z    +0.000, E1   +62.842, E3 +193188.160}
SPL {X  -149.257, Y  +328.060, Z    +0.000, E1   +62.292, E3 +193202.017}
SPL {X  -144.838, Y  +317.715, Z    +0.000, E1   +61.617, E3 +193217.023}
SPL {X  -139.661, Y  +307.631, Z    +0.000, E1   +60.727, E3 +193232.326}
SPL {X  -134.254, Y  +298.660, Z    +0.000, E1   +59.757, E3 +193246.374}
SPL {X  -111.782, Y  +271.224, Z    +0.000, E1   +50.030, E3 +193364.797}
ENDSPLINE

SPLINE
SPL {X  -142.230, Y  +312.416, Z    +0.000, E1   +39.081, E3 +193473.918}
SPL {X  -154.023, Y  +342.375, Z    +0.000, E1   +27.770, E3 +193490.375}
SPL {X  -159.227, Y  +369.989, Z    +0.000, E1   +12.792, E3 +193497.068}
SPL {X  -159.997, Y  +384.682, Z    +0.000, E1    +2.433, E3 +193498.432}
SPL {X  -160.000, Y  +388.025, Z    +0.000, E1    -0.434, E3 +193498.503}
SPL {X  -160.000, Y  +391.999, Z    +0.000, E1    -5.822, E3 +193498.647}
SPL {X  -160.000, Y  +397.968, Z    +0.000, E1   -15.492, E3 +193499.161}
SPL {X  -160.000, Y  +409.894, Z    +0.000, E1   -33.660, E3 +193501.269}
SPL {X  -160.000, Y  +457.050, Z    +0.000, E1   -59.500, E3 +193520.465}
SPL {X  -160.000, Y  +570.419, Z    +0.000, E1   -64.293, E3 +193606.030}
SPL {X  -160.000, Y  +587.690, Z    +0.000, E1   -64.299, E3 +193623.693}
SPL {X  -160.000, Y  +605.383, Z    +0.000, E1   -64.296, E3 +193641.791}
SPL {X  -160.000, Y  +621.010, Z    +0.000, E1   -64.279, E3 +193657.801}
SPL {X  -160.000, Y  +636.410, Z    +0.000, E1   -64.294, E3 +193673.530}
SPL {X  -160.000, Y  +654.238, Z    +0.000, E1   -64.301, E3 +193691.735}
SPL {X  -160.000, Y  +670.465, Z    +0.000, E1   -64.283, E3 +193708.359}
SPL {X  -159.617, Y  +685.462, Z    +0.000, E1   -64.244, E3 +193724.087}
SPL {X  -158.001, Y  +699.614, Z    +0.000, E1   -64.013, E3 +193740.261}
SPL {X  -155.628, Y  +711.546, Z    +0.000, E1   -63.666, E3 +193754.931}
SPL {X  -152.846, Y  +721.708, Z    +0.000, E1   -63.251, E3 +193768.163}
SPL {X  -149.418, Y  +731.620, Z    +0.000, E1   -62.736, E3 +193781.718}
SPL {X  -145.585, Y  +740.770, Z    +0.000, E1   -62.119, E3 +193794.817}
SPL {X  -141.572, Y  +748.948, Z    +0.000, E1   -61.453, E3 +193806.941}
SPL {X  -137.548, Y  +756.134, Z    +0.000, E1   -60.743, E3 +193817.950}
SPL {X  -133.391, Y  +762.756, Z    +0.000, E1   -59.994, E3 +193828.267}
SPL {X  -109.419, Y  +791.137, Z    +0.000, E1   -49.920, E3 +193961.556}
ENDSPLINE

SPLINE
SPL {X  -148.079, Y  +735.002, Z    +0.000, E1   -35.426, E3 +194069.139}
SPL {X  -158.158, Y  +698.608, Z    +0.000, E1   -18.222, E3 +194081.792}
SPL {X  -159.870, Y  +680.839, Z    +0.000, E1    -6.577, E3 +194084.179}
SPL {X  -160.000, Y  +671.754, Z    +0.000, E1    +0.400, E3 +194084.538}
SPL {X  -160.000, Y  +663.703, Z    +0.000, E1   +12.763, E3 +194085.004}
SPL {X  -160.000, Y  +653.310, Z    +0.000, E1   +30.441, E3 +194086.474}
SPL {X  -160.000, Y  +640.945, Z    +0.000, E1   +44.811, E3 +194089.686}
SPL {X  -160.000, Y  +592.314, Z    +0.000, E1   +61.740, E3 +194111.680}
SPL {X  -160.000, Y  +478.009, Z    +0.000, E1   +65.091, E3 +194198.737}
SPL {X  -160.000, Y  +417.917, Z    +0.000, E1   +69.146, E3 +194218.908}
SPL {X  -160.000, Y  +403.867, Z    +0.000, E1   +68.803, E3 +194233.400}
SPL {X  -160.000, Y  +399.669, Z    +0.000, E1   +67.598, E3 +194247.271}
SPL {X  -160.000, Y  +392.628, Z    +0.000, E1   +66.554, E3 +194262.302}
SPL {X  -159.998, Y  +384.859, Z    +0.000, E1   +65.356, E3 +194279.231}
SPL {X  -159.712, Y  +376.098, Z    +0.000, E1   +64.333, E3 +194295.775}
SPL {X  -158.506, Y  +363.887, Z    +0.000, E1   +63.706, E3 +194313.167}
SPL {X  -155.923, Y  +349.812, Z    +0.000, E1   +63.321, E3 +194330.520}
SPL {X  -152.732, Y  +338.026, Z    +0.000, E1   +62.842, E3 +194346.055}
SPL {X  -149.257, Y  +328.060, Z    +0.000, E1   +62.292, E3 +194359.911}
SPL {X  -144.838, Y  +317.715, Z    +0.000, E1   +61.617, E3 +194374.917}
SPL {X  -139.661, Y  +307.631, Z    +0.000, E1   +60.727, E3 +194390.220}
SPL {X  -134.254, Y  +298.660, Z    +0.000, E1   +59.757, E3 +194404.269}
SPL {X  -111.782, Y  +271.224, Z    +0.000, E1   +50.030, E3 +194522.692}
ENDSPLINE

SPLINE
SPL {X  -142.230, Y  +312.416, Z    +0.000, E1   +39.081, E3 +194631.812}
SPL {X  -154.023, Y  +342.375, Z    +0.000, E1   +27.770, E3 +194648.269}
SPL {X  -159.227, Y  +369.989, Z    +0.000, E1   +12.792, E3 +194654.962}
SPL {X  -159.997, Y  +384.682, Z    +0.000, E1    +2.433, E3 +194656.327}
SPL {X  -160.000, Y  +388.025, Z    +0.000, E1    -0.434, E3 +194656.397}
SPL {X  -160.000, Y  +391.999, Z    +0.000, E1    -5.822, E3 +194656.542}
SPL {X  -160.000, Y  +397.968, Z    +0.000, E1   -15.492, E3 +194657.056}
SPL {X  -160.000, Y  +409.894, Z    +0.000, E1   -33.660, E3 +194659.163}
SPL {X  -160.000, Y  +457.050, Z    +0.000, E1   -59.500, E3 +194678.360}
SPL {X  -160.000, Y  +570.419, Z    +0.000, E1   -64.293, E3 +194763.924}
SPL {X  -160.000, Y  +587.690, Z    +0.000, E1   -64.299, E3 +194781.587}
SPL {X  -160.000, Y  +605.383, Z    +0.000, E1   -64.296, E3 +194799.685}
SPL {X  -160.000, Y  +621.010, Z    +0.000, E1   -64.279, E3 +194815.695}
SPL {X  -160.000, Y  +636.410, Z    +0.000, E1   -64.294, E3 +194831.424}
SPL {X  -160.000, Y  +654.238, Z    +0.000, E1   -64.301, E3 +194849.630}
SPL {X  -160.000, Y  +670.465, Z    +0.000, E1   -64.283, E3 +194866.253}
SPL {X  -159.617, Y  +685.462, Z    +0.000, E1   -64.244, E3 +194881.981}
SPL {X  -158.001, Y  +699.614, Z    +0.000, E1   -64.013, E3 +194898.156}
SPL {X  -155.628, Y  +711.546, Z    +0.000, E1   -63.666, E3 +194912.825}
SPL {X  -152.846, Y  +721.708, Z    +0.000, E1   -63.251, E3 +194926.058}
SPL {X  -149.418, Y  +731.620, Z    +0.000, E1   -62.736, E3 +194939.612}
SPL {X  -145.585, Y  +740.770, Z    +0.000, E1   -62.119, E3 +194952.711}
SPL {X  -141.572, Y  +748.948, Z    +0.000, E1   -61.453, E3 +194964.835}
SPL {X  -137.548, Y  +756.134, Z    +0.000, E1   -60.743, E3 +194975.845}
SPL {X  -133.391, Y  +762.756, Z    +0.000, E1   -59.994, E3 +194986.161}
SPL {X  -109.419, Y  +791.137, Z    +0.000, E1   -49.920, E3 +195119.450}
ENDSPLINE

SPLINE
SPL {X  -148.079, Y  +735.002, Z    +0.000, E1   -35.426, E3 +195227.033}
SPL {X  -158.158, Y  +698.608, Z    +0.000, E1   -18.222, E3 +195239.686}
SPL {X  -159.870, Y  +680.839, Z    +0.000, E1    -6.577, E3 +195242.074}
SPL {X  -160.000, Y  +671.754, Z    +0.000, E1    +0.400, E3 +195242.432}
SPL {X  -160.000, Y  +663.703, Z    +0.000, E1   +12.763, E3 +195242.898}
SPL {X  -160.000, Y  +653.310, Z    +0.000, E1   +30.441, E3 +195244.368}
SPL {X  -160.000, Y  +640.945, Z    +0.000, E1   +44.811, E3 +195247.580}
SPL {X  -160.000, Y  +592.314, Z    +0.000, E1   +61.740, E3 +195269.574}
SPL {X  -160.000, Y  +478.009, Z    +0.000, E1   +65.091, E3 +195356.632}
SPL {X  -160.000, Y  +417.917, Z    +0.000, E1   +69.146, E3 +195376.802}
SPL {X  -160.000, Y  +403.867, Z    +0.000, E1   +68.803, E3 +195391.295}
SPL {X  -160.000, Y  +399.669, Z    +0.000, E1   +67.598, E3 +195405.166}
SPL {X  -160.000, Y  +392.628, Z    +0.000, E1   +66.554, E3 +195420.197}
SPL {X  -159.998, Y  +384.859, Z    +0.000, E1   +65.356, E3 +195437.125}
SPL {X  -159.712, Y  +376.098, Z    +0.000, E1   +64.333, E3 +195453.669}
SPL {X  -158.506, Y  +363.887, Z    +0.000, E1   +63.706, E3 +195471.061}
SPL {X  -155.923, Y  +349.812, Z    +0.000, E1   +63.321, E3 +195488.415}
SPL {X  -152.732, Y  +338.026, Z    +0.000, E1   +62.842, E3 +195503.949}
SPL {X  -149.257, Y  +328.060, Z    +0.000, E1   +62.292, E3 +195517.806}
SPL {X  -144.838, Y  +317.715, Z    +0.000, E1   +61.617, E3 +195532.812}
SPL {X  -139.661, Y  +307.631, Z    +0.000, E1   +60.727, E3 +195548.115}
SPL {X  -134.254, Y  +298.660, Z    +0.000, E1   +59.757, E3 +195562.163}
SPL {X  -111.782, Y  +271.224, Z    +0.000, E1   +50.030, E3 +195680.586}
ENDSPLINE

SPLINE
SPL {X  -142.230, Y  +312.416, Z    +0.000, E1   +39.081, E3 +195789.706}
SPL {X  -154.023, Y  +342.375, Z    +0.000, E1   +27.770, E3 +195806.163}
SPL {X  -159.227, Y  +369.989, Z    +0.000, E1   +12.792, E3 +195812.856}
SPL {X  -159.997, Y  +384.682, Z    +0.000, E1    +2.433, E3 +195814.221}
SPL {X  -160.000, Y  +388.025, Z    +0.000, E1    -0.434, E3 +195814.291}
SPL {X  -160.000, Y  +391.999, Z    +0.000, E1    -5.822, E3 +195814.436}
SPL {X  -160.000, Y  +397.968, Z    +0.000, E1   -15.492, E3 +195814.950}
SPL {X  -160.000, Y  +409.894, Z    +0.000, E1   -33.660, E3 +195817.057}
SPL {X  -160.000, Y  +457.050, Z    +0.000, E1   -59.500, E3 +195836.254}
SPL {X  -160.000, Y  +570.419, Z    +0.000, E1   -64.293, E3 +195921.819}
SPL {X  -160.000, Y  +587.690, Z    +0.000, E1   -64.299, E3 +195939.481}
SPL {X  -160.000, Y  +605.383, Z    +0.000, E1   -64.296, E3 +195957.580}
SPL {X  -160.000, Y  +621.010, Z    +0.000, E1   -64.279, E3 +195973.590}
SPL {X  -160.000, Y  +636.410, Z    +0.000, E1   -64.294, E3 +195989.318}
SPL {X  -160.000, Y  +654.238, Z    +0.000, E1   -64.301, E3 +196007.524}
SPL {X  -160.000, Y  +670.465, Z    +0.000, E1   -64.283, E3 +196024.147}
SPL {X  -159.617, Y  +685.462, Z    +0.000, E1   -64.244, E3 +196039.875}
SPL {X  -158.001, Y  +699.614, Z    +0.000, E1   -64.013, E3 +196056.050}
SPL {X  -155.628, Y  +711.546, Z    +0.000, E1   -63.666, E3 +196070.719}
SPL {X  -152.846, Y  +721.708, Z    +0.000, E1   -63.251, E3 +196083.952}
SPL {X  -149.418, Y  +731.620, Z    +0.000, E1   -62.736, E3 +196097.507}
SPL {X  -145.585, Y  +740.770, Z    +0.000, E1   -62.119, E3 +196110.605}
SPL {X  -141.572, Y  +748.948, Z    +0.000, E1   -61.453, E3 +196122.729}
SPL {X  -137.548, Y  +756.134, Z    +0.000, E1   -60.743, E3 +196133.739}
SPL {X  -133.391, Y  +762.756, Z    +0.000, E1   -59.994, E3 +196144.056}
SPL {X  -109.419, Y  +791.137, Z    +0.000, E1   -49.920, E3 +196277.345}
ENDSPLINE

SPLINE
SPL {X  -148.079, Y  +735.002, Z    +0.000, E1   -35.426, E3 +196384.927}
SPL {X  -158.158, Y  +698.608, Z    +0.000, E1   -18.222, E3 +196397.580}
SPL {X  -159.870, Y  +680.839, Z    +0.000, E1    -6.577, E3 +196399.968}
SPL {X  -160.000, Y  +671.754, Z    +0.000, E1    +0.400, E3 +196400.327}
SPL {X  -160.000, Y  +663.703, Z    +0.000, E1   +12.763, E3 +196400.792}
SPL {X  -160.000, Y  +653.310, Z    +0.000, E1   +30.441, E3 +196402.263}
SPL {X  -160.000, Y  +640.945, Z    +0.000, E1   +44.811, E3 +196405.475}
SPL {X  -160.000, Y  +592.314, Z    +0.000, E1   +61.740, E3 +196427.468}
SPL {X  -160.000, Y  +478.009, Z    +0.000, E1   +65.091, E3 +196514.526}
SPL {X  -160.000, Y  +417.917, Z    +0.000, E1   +69.146, E3 +196534.696}
SPL {X  -160.000, Y  +403.867, Z    +0.000, E1   +68.803, E3 +196549.189}
SPL {X  -160.000, Y  +399.669, Z    +0.000, E1   +67.598, E3 +196563.060}
SPL {X  -160.000, Y  +392.628, Z    +0.000, E1   +66.554, E3 +196578.091}
SPL {X  -159.998, Y  +384.859, Z    +0.000, E1   +65.356, E3 +196595.019}
SPL {X  -159.712, Y  +376.098, Z    +0.000, E1   +64.333, E3 +196611.564}
ENDSPLINE

SPLINE
SPL {X  -159.744, Y  +376.651, Z    +0.000, E1   +61.772, E3 +196629.948}
SPL {X  -158.128, Y  +361.299, Z    +0.000, E1   +61.520, E3 +196649.167}
SPL {X  -155.661, Y  +348.690, Z    +0.000, E1   +61.132, E3 +196666.123}
SPL {X  -152.251, Y  +336.510, Z    +0.000, E1   +60.617, E3 +196683.456}
SPL {X  -148.078, Y  +325.096, Z    +0.000, E1   +59.928, E3 +196700.584}
SPL {X  -143.290, Y  +314.510, Z    +0.000, E1   +59.129, E3 +196717.207}
SPL {X  -139.113, Y  +306.659, Z    +0.000, E1   +58.310, E3 +196730.058}
SPL {X  -135.700, Y  +300.932, Z    +0.000, E1   +57.683, E3 +196739.554}
SPL {X  -117.539, Y  +277.143, Z    +0.000, E1   +48.559, E3 +196854.240}
ENDSPLINE

SPLINE
SPL {X  -150.734, Y  +332.041, Z    +0.000, E1   +31.286, E3 +196956.905}
SPL {X  -159.235, Y  +370.077, Z    +0.000, E1   +12.240, E3 +196970.259}
SPL {X  -159.991, Y  +384.025, Z    +0.000, E1    +2.884, E3 +196971.808}
SPL {X  -160.000, Y  +388.170, Z    +0.000, E1    -0.470, E3 +196971.939}
SPL {X  -160.000, Y  +392.385, Z    +0.000, E1    -5.697, E3 +196972.129}
SPL {X  -160.000, Y  +398.918, Z    +0.000, E1   -15.420, E3 +196972.807}
SPL {X  -160.000, Y  +410.991, Z    +0.000, E1   -32.499, E3 +196975.302}
SPL {X  -160.000, Y  +455.466, Z    +0.000, E1   -56.407, E3 +196996.201}
SPL {X  -160.000, Y  +554.875, Z    +0.000, E1   -61.915, E3 +197078.105}
SPL {X  -160.000, Y  +571.700, Z    +0.000, E1   -61.918, E3 +197097.182}
SPL {X  -160.000, Y  +587.975, Z    +0.000, E1   -61.909, E3 +197115.648}
SPL {X  -160.000, Y  +604.690, Z    +0.000, E1   -61.922, E3 +197134.578}
SPL {X  -160.000, Y  +621.475, Z    +0.000, E1   -61.913, E3 +197153.630}
SPL {X  -160.000, Y  +638.005, Z    +0.000, E1   -61.917, E3 +197172.360}
SPL {X  -160.000, Y  +655.083, Z    +0.000, E1   -61.921, E3 +197191.721}
SPL {X  -160.000, Y  +671.910, Z    +0.000, E1   -61.915, E3 +197210.815}
SPL {X  -159.476, Y  +687.338, Z    +0.000, E1   -61.835, E3 +197228.867}
SPL {X  -157.928, Y  +700.064, Z    +0.000, E1   -61.593, E3 +197244.932}
SPL {X  -155.236, Y  +713.154, Z    +0.000, E1   -61.225, E3 +197262.479}
SPL {X  -151.860, Y  +724.785, Z    +0.000, E1   -60.654, E3 +197279.151}
SPL {X  -148.451, Y  +734.085, Z    +0.000, E1   -60.099, E3 +197293.077}
SPL {X  -144.033, Y  +744.073, Z    +0.000, E1   -59.381, E3 +197308.597}
SPL {X  -139.170, Y  +753.341, Z    +0.000, E1   -58.489, E3 +197323.618}
SPL {X  -135.320, Y  +759.772, Z    +0.000, E1   -57.727, E3 +197334.328}
SPL {X  -117.185, Y  +783.339, Z    +0.000, E1   -48.966, E3 +197442.714}
ENDSPLINE

SPLINE
SPL {X  -142.074, Y  +747.987, Z    +0.000, E1   -38.326, E3 +197541.408}
SPL {X  -154.075, Y  +717.539, Z    +0.000, E1   -26.988, E3 +197560.565}
SPL {X  -158.904, Y  +693.092, Z    +0.000, E1   -14.171, E3 +197567.356}
SPL {X  -159.937, Y  +678.885, Z    +0.000, E1    -4.971, E3 +197569.183}
SPL {X  -160.000, Y  +672.790, Z    +0.000, E1    -0.387, E3 +197569.451}
SPL {X  -160.000, Y  +669.961, Z    +0.000, E1    +2.696, E3 +197569.528}
SPL {X  -160.000, Y  +663.591, Z    +0.000, E1   +11.688, E3 +197570.022}
SPL {X  -160.000, Y  +654.521, Z    +0.000, E1   +25.997, E3 +197571.380}
SPL {X  -160.000, Y  +642.364, Z    +0.000, E1   +40.387, E3 +197574.682}
SPL {X  -160.000, Y  +597.330, Z    +0.000, E1   +58.145, E3 +197597.593}
SPL {X  -160.000, Y  +507.195, Z    +0.000, E1   +61.792, E3 +197674.924}
SPL {X  -160.000, Y  +494.139, Z    +0.000, E1   +61.770, E3 +197689.854}
SPL {X  -160.000, Y  +480.560, Z    +0.000, E1   +61.503, E3 +197707.651}
ENDSPLINE

SPLINE
SPL {X  -160.000, Y  +495.136, Z    +0.000, E1   +55.416, E3 +197729.158}
ENDSPLINE

SPLINE
SPL {X  -160.000, Y  +472.196, Z    +0.000, E1   +56.977, E3 +197751.833}
SPL {X  -160.000, Y  +448.172, Z    +0.000, E1   +58.434, E3 +197774.528}
SPL {X  -160.000, Y  +423.986, Z    +0.000, E1   +59.836, E3 +197795.781}
SPL {X  -160.000, Y  +398.875, Z    +0.000, E1   +61.100, E3 +197817.329}
SPL {X  -159.733, Y  +376.466, Z    +0.000, E1   +61.765, E3 +197838.519}
SPL {X  -158.128, Y  +361.299, Z    +0.000, E1   +61.520, E3 +197857.499}
SPL {X  -155.661, Y  +348.690, Z    +0.000, E1   +61.132, E3 +197874.455}
SPL {X  -152.251, Y  +336.510, Z    +0.000, E1   +60.617, E3 +197891.787}
SPL {X  -148.078, Y  +325.096, Z    +0.000, E1   +59.928, E3 +197908.916}
SPL {X  -143.290, Y  +314.510, Z    +0.000, E1   +59.129, E3 +197925.539}
SPL {X  -139.113, Y  +306.659, Z    +0.000, E1   +58.310, E3 +197938.389}
SPL {X  -135.700, Y  +300.932, Z    +0.000, E1   +57.683, E3 +197947.886}
SPL {X  -117.539, Y  +277.143, Z    +0.000, E1   +48.559, E3 +198062.572}
ENDSPLINE

SPLINE
SPL {X  -150.734, Y  +332.041, Z    +0.000, E1   +31.286, E3 +198165.237}
SPL {X  -159.235, Y  +370.077, Z    +0.000, E1   +12.240, E3 +198178.591}
SPL {X  -159.991, Y  +384.025, Z    +0.000, E1    +2.884, E3 +198180.140}
SPL {X  -160.000, Y  +388.170, Z    +0.000, E1    -0.470, E3 +198180.270}
SPL {X  -160.000, Y  +392.385, Z    +0.000, E1    -5.697, E3 +198180.460}
SPL {X  -160.000, Y  +398.918, Z    +0.000, E1   -15.420, E3 +198181.139}
SPL {X  -160.000, Y  +410.991, Z    +0.000, E1   -32.499, E3 +198183.634}
SPL {X  -160.000, Y  +455.466, Z    +0.000, E1   -56.407, E3 +198204.533}
SPL {X  -160.000, Y  +554.875, Z    +0.000, E1   -61.915, E3 +198286.437}
SPL {X  -160.000, Y  +571.700, Z    +0.000, E1   -61.918, E3 +198305.514}
SPL {X  -160.000, Y  +587.975, Z    +0.000, E1   -61.909, E3 +198323.980}
SPL {X  -160.000, Y  +604.690, Z    +0.000, E1   -61.922, E3 +198342.910}
SPL {X  -160.000, Y  +621.475, Z    +0.000, E1   -61.913, E3 +198361.961}
SPL {X  -160.000, Y  +638.005, Z    +0.000, E1   -61.917, E3 +198380.692}
SPL {X  -160.000, Y  +655.083, Z    +0.000, E1   -61.921, E3 +198400.053}
SPL {X  -160.000, Y  +671.910, Z    +0.000, E1   -61.915, E3 +198419.147}
SPL {X  -159.476, Y  +687.338, Z    +0.000, E1   -61.835, E3 +198437.199}
SPL {X  -157.928, Y  +700.064, Z    +0.000, E1   -61.593, E3 +198453.263}
SPL {X  -155.236, Y  +713.154, Z    +0.000, E1   -61.225, E3 +198470.811}
SPL {X  -151.860, Y  +724.785, Z    +0.000, E1   -60.654, E3 +198487.483}
SPL {X  -148.451, Y  +734.085, Z    +0.000, E1   -60.099, E3 +198501.408}
SPL {X  -144.033, Y  +744.073, Z    +0.000, E1   -59.381, E3 +198516.929}
SPL {X  -139.170, Y  +753.341, Z    +0.000, E1   -58.489, E3 +198531.950}
SPL {X  -135.320, Y  +759.772, Z    +0.000, E1   -57.727, E3 +198542.660}
SPL {X  -117.185, Y  +783.339, Z    +0.000, E1   -48.966, E3 +198651.046}
ENDSPLINE

SPLINE
SPL {X  -142.074, Y  +747.987, Z    +0.000, E1   -38.326, E3 +198749.740}
SPL {X  -154.075, Y  +717.539, Z    +0.000, E1   -26.988, E3 +198768.897}
SPL {X  -158.904, Y  +693.092, Z    +0.000, E1   -14.171, E3 +198775.688}
SPL {X  -159.937, Y  +678.885, Z    +0.000, E1    -4.971, E3 +198777.515}
SPL {X  -160.000, Y  +672.790, Z    +0.000, E1    -0.387, E3 +198777.783}
SPL {X  -160.000, Y  +669.961, Z    +0.000, E1    +2.696, E3 +198777.860}
SPL {X  -160.000, Y  +663.591, Z    +0.000, E1   +11.688, E3 +198778.354}
SPL {X  -160.000, Y  +654.521, Z    +0.000, E1   +25.997, E3 +198779.712}
SPL {X  -160.000, Y  +642.364, Z    +0.000, E1   +40.387, E3 +198783.014}
SPL {X  -160.000, Y  +597.330, Z    +0.000, E1   +58.145, E3 +198805.925}
SPL {X  -160.000, Y  +507.195, Z    +0.000, E1   +61.792, E3 +198883.256}
SPL {X  -160.000, Y  +494.139, Z    +0.000, E1   +61.770, E3 +198898.186}
SPL {X  -160.000, Y  +480.560, Z    +0.000, E1   +61.503, E3 +198915.983}
ENDSPLINE

SPLINE
SPL {X  -160.000, Y  +495.136, Z    +0.000, E1   +55.416, E3 +198937.490}
ENDSPLINE

SPLINE
SPL {X  -160.000, Y  +472.196, Z    +0.000, E1   +56.977, E3 +198960.165}
SPL {X  -160.000, Y  +448.172, Z    +0.000, E1   +58.434, E3 +198982.859}
SPL {X  -160.000, Y  +423.986, Z    +0.000, E1   +59.836, E3 +199004.113}
SPL {X  -160.000, Y  +398.875, Z    +0.000, E1   +61.100, E3 +199025.661}
SPL {X  -159.733, Y  +376.466, Z    +0.000, E1   +61.765, E3 +199046.851}
SPL {X  -158.128, Y  +361.299, Z    +0.000, E1   +61.520, E3 +199065.830}
SPL {X  -155.661, Y  +348.690, Z    +0.000, E1   +61.132, E3 +199082.786}
SPL {X  -152.251, Y  +336.510, Z    +0.000, E1   +60.617, E3 +199100.119}
SPL {X  -148.078, Y  +325.096, Z    +0.000, E1   +59.928, E3 +199117.248}
SPL {X  -143.290, Y  +314.510, Z    +0.000, E1   +59.129, E3 +199133.870}
SPL {X  -139.113, Y  +306.659, Z    +0.000, E1   +58.310, E3 +199146.721}
SPL {X  -135.700, Y  +300.932, Z    +0.000, E1   +57.683, E3 +199156.218}
SPL {X  -117.539, Y  +277.143, Z    +0.000, E1   +48.559, E3 +199270.904}
ENDSPLINE

SPLINE
SPL {X  -150.734, Y  +332.041, Z    +0.000, E1   +31.286, E3 +199373.568}
SPL {X  -159.235, Y  +370.077, Z    +0.000, E1   +12.240, E3 +199386.923}
SPL {X  -159.991, Y  +384.025, Z    +0.000, E1    +2.884, E3 +199388.471}
SPL {X  -160.000, Y  +388.170, Z    +0.000, E1    -0.470, E3 +199388.602}
SPL {X  -160.000, Y  +392.385, Z    +0.000, E1    -5.697, E3 +199388.792}
SPL {X  -160.000, Y  +398.918, Z    +0.000, E1   -15.420, E3 +199389.471}
SPL {X  -160.000, Y  +410.991, Z    +0.000, E1   -32.499, E3 +199391.966}
SPL {X  -160.000, Y  +455.466, Z    +0.000, E1   -56.407, E3 +199412.865}
SPL {X  -160.000, Y  +554.875, Z    +0.000, E1   -61.915, E3 +199494.769}
SPL {X  -160.000, Y  +571.700, Z    +0.000, E1   -61.918, E3 +199513.845}
SPL {X  -160.000, Y  +587.975, Z    +0.000, E1   -61.909, E3 +199532.312}
SPL {X  -160.000, Y  +604.690, Z    +0.000, E1   -61.922, E3 +199551.241}
SPL {X  -160.000, Y  +621.475, Z    +0.000, E1   -61.913, E3 +199570.293}
SPL {X  -160.000, Y  +638.005, Z    +0.000, E1   -61.917, E3 +199589.024}
SPL {X  -160.000, Y  +655.083, Z    +0.000, E1   -61.921, E3 +199608.385}
SPL {X  -160.000, Y  +671.910, Z    +0.000, E1   -61.915, E3 +199627.479}
SPL {X  -159.476, Y  +687.338, Z    +0.000, E1   -61.835, E3 +199645.531}
SPL {X  -157.928, Y  +700.064, Z    +0.000, E1   -61.593, E3 +199661.595}
SPL {X  -155.236, Y  +713.154, Z    +0.000, E1   -61.225, E3 +199679.142}
SPL {X  -151.860, Y  +724.785, Z    +0.000, E1   -60.654, E3 +199695.815}
SPL {X  -148.451, Y  +734.085, Z    +0.000, E1   -60.099, E3 +199709.740}
SPL {X  -144.033, Y  +744.073, Z    +0.000, E1   -59.381, E3 +199725.260}
SPL {X  -139.170, Y  +753.341, Z    +0.000, E1   -58.489, E3 +199740.282}
SPL {X  -135.320, Y  +759.772, Z    +0.000, E1   -57.727, E3 +199750.992}
SPL {X  -117.185, Y  +783.339, Z    +0.000, E1   -48.966, E3 +199859.378}
ENDSPLINE

SPLINE
SPL {X  -142.074, Y  +747.987, Z    +0.000, E1   -38.326, E3 +199958.071}
SPL {X  -154.075, Y  +717.539, Z    +0.000, E1   -26.988, E3 +199977.228}
SPL {X  -158.904, Y  +693.092, Z    +0.000, E1   -14.171, E3 +199984.019}
SPL {X  -159.937, Y  +678.885, Z    +0.000, E1    -4.971, E3 +199985.847}
SPL {X  -160.000, Y  +672.790, Z    +0.000, E1    -0.387, E3 +199986.115}
SPL {X  -160.000, Y  +669.961, Z    +0.000, E1    +2.696, E3 +199986.191}
SPL {X  -160.000, Y  +663.591, Z    +0.000, E1   +11.688, E3 +199986.686}
SPL {X  -160.000, Y  +654.521, Z    +0.000, E1   +25.997, E3 +199988.043}
SPL {X  -160.000, Y  +642.364, Z    +0.000, E1   +40.387, E3 +199991.346}
SPL {X  -160.000, Y  +597.330, Z    +0.000, E1   +58.145, E3 +200014.257}
SPL {X  -160.000, Y  +507.195, Z    +0.000, E1   +61.792, E3 +200091.588}
SPL {X  -160.000, Y  +494.139, Z    +0.000, E1   +61.770, E3 +200106.518}
SPL {X  -160.000, Y  +480.560, Z    +0.000, E1   +61.503, E3 +200124.315}
ENDSPLINE

SPLINE
SPL {X  -160.000, Y  +495.136, Z    +0.000, E1   +55.416, E3 +200145.822}
ENDSPLINE

SPLINE
SPL {X  -160.000, Y  +472.196, Z    +0.000, E1   +56.977, E3 +200168.497}
SPL {X  -160.000, Y  +448.172, Z    +0.000, E1   +58.434, E3 +200191.191}
SPL {X  -160.000, Y  +423.986, Z    +0.000, E1   +59.836, E3 +200212.445}
SPL {X  -160.000, Y  +398.875, Z    +0.000, E1   +61.100, E3 +200233.993}
SPL {X  -159.733, Y  +376.466, Z    +0.000, E1   +61.765, E3 +200255.182}
SPL {X  -158.128, Y  +361.299, Z    +0.000, E1   +61.520, E3 +200274.162}
SPL {X  -155.661, Y  +348.690, Z    +0.000, E1   +61.132, E3 +200291.118}
SPL {X  -152.251, Y  +336.510, Z    +0.000, E1   +60.617, E3 +200308.451}
SPL {X  -148.078, Y  +325.096, Z    +0.000, E1   +59.928, E3 +200325.579}
SPL {X  -143.290, Y  +314.510, Z    +0.000, E1   +59.129, E3 +200342.202}
SPL {X  -139.113, Y  +306.659, Z    +0.000, E1   +58.310, E3 +200355.053}
SPL {X  -135.700, Y  +300.932, Z    +0.000, E1   +57.683, E3 +200364.550}
SPL {X  -117.539, Y  +277.143, Z    +0.000, E1   +48.559, E3 +200479.236}
ENDSPLINE

SPLINE
SPL {X  -150.734, Y  +332.041, Z    +0.000, E1   +31.286, E3 +200581.900}
SPL {X  -159.235, Y  +370.077, Z    +0.000, E1   +12.240, E3 +200595.254}
SPL {X  -159.991, Y  +384.025, Z    +0.000, E1    +2.884, E3 +200596.803}
SPL {X  -160.000, Y  +388.170, Z    +0.000, E1    -0.470, E3 +200596.934}
SPL {X  -160.000, Y  +392.385, Z    +0.000, E1    -5.697, E3 +200597.124}
SPL {X  -160.000, Y  +398.918, Z    +0.000, E1   -15.420, E3 +200597.802}
SPL {X  -160.000, Y  +410.991, Z    +0.000, E1   -32.499, E3 +200600.298}
SPL {X  -160.000, Y  +455.466, Z    +0.000, E1   -56.407, E3 +200621.196}
SPL {X  -160.000, Y  +554.875, Z    +0.000, E1   -61.915, E3 +200703.100}
SPL {X  -160.000, Y  +571.700, Z    +0.000, E1   -61.918, E3 +200722.177}
SPL {X  -160.000, Y  +587.975, Z    +0.000, E1   -61.909, E3 +200740.644}
SPL {X  -160.000, Y  +604.690, Z    +0.000, E1   -61.922, E3 +200759.573}
SPL {X  -160.000, Y  +621.475, Z    +0.000, E1   -61.913, E3 +200778.625}
SPL {X  -160.000, Y  +638.005, Z    +0.000, E1   -61.917, E3 +200797.355}
SPL {X  -160.000, Y  +655.083, Z    +0.000, E1   -61.921, E3 +200816.717}
SPL {X  -160.000, Y  +671.910, Z    +0.000, E1   -61.915, E3 +200835.811}
SPL {X  -159.476, Y  +687.338, Z    +0.000, E1   -61.835, E3 +200853.863}
SPL {X  -157.928, Y  +700.064, Z    +0.000, E1   -61.593, E3 +200869.927}
SPL {X  -155.236, Y  +713.154, Z    +0.000, E1   -61.225, E3 +200887.474}
SPL {X  -151.860, Y  +724.785, Z    +0.000, E1   -60.654, E3 +200904.147}
SPL {X  -148.451, Y  +734.085, Z    +0.000, E1   -60.099, E3 +200918.072}
SPL {X  -144.033, Y  +744.073, Z    +0.000, E1   -59.381, E3 +200933.592}
SPL {X  -139.170, Y  +753.341, Z    +0.000, E1   -58.489, E3 +200948.614}
SPL {X  -135.320, Y  +759.772, Z    +0.000, E1   -57.727, E3 +200959.323}
SPL {X  -117.185, Y  +783.339, Z    +0.000, E1   -48.966, E3 +201067.709}
ENDSPLINE

SPLINE
SPL {X  -142.074, Y  +747.987, Z    +0.000, E1   -38.326, E3 +201166.403}
SPL {X  -154.075, Y  +717.539, Z    +0.000, E1   -26.988, E3 +201185.560}
SPL {X  -158.904, Y  +693.092, Z    +0.000, E1   -14.171, E3 +201192.351}
SPL {X  -159.937, Y  +678.885, Z    +0.000, E1    -4.971, E3 +201194.178}
SPL {X  -160.000, Y  +672.790, Z    +0.000, E1    -0.387, E3 +201194.446}
SPL {X  -160.000, Y  +669.961, Z    +0.000, E1    +2.696, E3 +201194.523}
SPL {X  -160.000, Y  +663.591, Z    +0.000, E1   +11.688, E3 +201195.017}
SPL {X  -160.000, Y  +654.521, Z    +0.000, E1   +25.997, E3 +201196.375}
SPL {X  -160.000, Y  +642.364, Z    +0.000, E1   +40.387, E3 +201199.677}
SPL {X  -160.000, Y  +597.330, Z    +0.000, E1   +58.145, E3 +201222.588}
SPL {X  -160.000, Y  +507.195, Z    +0.000, E1   +61.792, E3 +201299.919}
SPL {X  -160.000, Y  +494.139, Z    +0.000, E1   +61.770, E3 +201314.850}
SPL {X  -160.000, Y  +480.560, Z    +0.000, E1   +61.503, E3 +201332.647}
ENDSPLINE

SPLINE
SPL {X  -160.000, Y  +495.136, Z    +0.000, E1   +55.416, E3 +201354.153}
ENDSPLINE

